LIN {X 0,Y 256.355,Z 531.803,A -85,B 0,C 180,E1 -21459.86,E2 -21459.86} C_VEL
LIN {X 0,Y 252.646,Z 547.764,A -85,B 0,C 180,E1 -21461.014,E2 -21461.014} C_VEL
LIN {X 0,Y 248.399,Z 562.44,A -85,B 0,C 180,E1 -21462.341,E2 -21462.341} C_VEL
LIN {X 0,Y 243.325,Z 577.415,A -85,B 0,C 180,E1 -21464.072,E2 -21464.072} C_VEL
LIN {X 0,Y 238.018,Z 591.108,A -85,B 0,C 180,E1 -21466.062,E2 -21466.062} C_VEL
LIN {X 0,Y 233.373,Z 601.837,A -85,B 0,C 180,E1 -21467.929,E2 -21467.929} C_VEL
LIN {X 0,Y 227.446,Z 614.36,A -85,B 0,C 180,E1 -21470.578,E2 -21470.578} C_VEL
LIN {X 0,Y 221.787,Z 625.54,A -85,B 0,C 180,E1 -21473.548,E2 -21473.548} C_VEL
LIN {X 0,Y 216.728,Z 634.804,A -85,B 0,C 180,E1 -21476.546,E2 -21476.546} C_VEL
LIN {X 0,Y 211.759,Z 643.811,A -85,B 0,C 180,E1 -21480.144,E2 -21480.144} C_VEL
LIN {X 0,Y 207.469,Z 651.338,A -85,B 0,C 180,E1 -21483.872,E2 -21483.872} C_VEL
LIN {X 0,Y 204.013,Z 657.483,A -85,B 0,C 180,E1 -21487.732,E2 -21487.732} C_VEL
LIN {X 0,Y 201.336,Z 662.513,A -85,B 0,C 180,E1 -21491.69,E2 -21491.69} C_VEL
LIN {X 0,Y 199.353,Z 666.403,A -85,B 0,C 180,E1 -21495.713,E2 -21495.713} C_VEL
LIN {X 0,Y 198.192,Z 669.285,A -85,B 0,C 180,E1 -21499.787,E2 -21499.787} C_VEL
LIN {X 0,Y 197.545,Z 671.175,A -85,B 0,C 180,E1 -21503.873,E2 -21503.873} C_VEL
LIN {X 0,Y 197.351,Z 672.126,A -85,B 0,C 180,E1 -21507.959,E2 -21507.959} C_VEL
LIN {X 0,Y 197.395,Z 672.279,A -85,B 0,C 180,E1 -21510,E2 -21510} C_VEL
LIN {X 0,Y 197.415,Z 671.675,A -85,B 0,C 180,E1 -21514.579,E2 -21514.579} C_VEL
LIN {X 0,Y 197.782,Z 670.45,A -85,B 0,C 180,E1 -21518.171,E2 -21518.171} C_VEL
LIN {X 0,Y 198.684,Z 668.056,A -85,B 0,C 180,E1 -21522.253,E2 -21522.253} C_VEL
LIN {X 0,Y 200.261,Z 664.751,A -85,B 0,C 180,E1 -21526.305,E2 -21526.305} C_VEL
LIN {X 0,Y 203.161,Z 659.194,A -85,B 0,C 180,E1 -21531.192,E2 -21531.192} C_VEL
LIN {X 0,Y 207.427,Z 651.578,A -85,B 0,C 180,E1 -21536.133,E2 -21536.133} C_VEL
LIN {X 0,Y 212.494,Z 642.647,A -85,B 0,C 180,E1 -21540.524,E2 -21540.524} C_VEL
LIN {X 0,Y 217.342,Z 633.912,A -85,B 0,C 180,E1 -21543.903,E2 -21543.903} C_VEL
LIN {X 0,Y 222.404,Z 624.465,A -85,B 0,C 180,E1 -21546.898,E2 -21546.898} C_VEL
LIN {X 0,Y 227.991,Z 613.516,A -85,B 0,C 180,E1 -21549.74,E2 -21549.74} C_VEL
LIN {X 0,Y 234.118,Z 600.392,A -85,B 0,C 180,E1 -21552.487,E2 -21552.487} C_VEL
LIN {X 0,Y 240.281,Z 586.013,A -85,B 0,C 180,E1 -21554.847,E2 -21554.847} C_VEL
LIN {X 0,Y 245.182,Z 572.494,A -85,B 0,C 180,E1 -21556.664,E2 -21556.664} C_VEL
LIN {X 0,Y 249.822,Z 558.149,A -85,B 0,C 180,E1 -21558.201,E2 -21558.201} C_VEL
LIN {X 0,Y 254.135,Z 542.579,A -85,B 0,C 180,E1 -21559.508,E2 -21559.508} C_VEL
LIN {X 0,Y 257.325,Z 527.974,A -85,B 0,C 180,E1 -21560.493,E2 -21560.493} C_VEL
LIN {X 0,Y 259.966,Z 512.67,A -85,B 0,C 180,E1 -21561.239,E2 -21561.239} C_VEL
LIN {X 0,Y 261.928,Z 495.841,A -85,B 0,C 180,E1 -21561.832,E2 -21561.832} C_VEL
LIN {X 0,Y 268.666,Z 399.885,A -85,B 0,C 180,E1 -21564.176,E2 -21564.176} C_VEL
LIN {X 0,Y 261.466,Z 386.886,A -85,B 0,C 180,E1 -21567.08,E2 -21567.08} C_VEL
LIN {X 0,Y 255.056,Z 376.394,A -85,B 0,C 180,E1 -21569.969,E2 -21569.969} C_VEL
LIN {X 0,Y 249.229,Z 367.595,A -85,B 0,C 180,E1 -21572.938,E2 -21572.938} C_VEL
LIN {X 0,Y 243.586,Z 359.592,A -85,B 0,C 180,E1 -21576.259,E2 -21576.259} C_VEL
LIN {X 0,Y 240.202,Z 355.081,A -85,B 0,C 180,E1 -21578.547,E2 -21578.547} C_VEL
LIN {X 0,Y 237.313,Z 351.233,A -85,B 0,C 180,E1 -21580.763,E2 -21580.763} C_VEL
LIN {X 0,Y 233.816,Z 346.937,A -85,B 0,C 180,E1 -21583.889,E2 -21583.889} C_VEL
LIN {X 0,Y 233.178,Z 345.639,A -85,B 0,C 180,E1 -21584.597,E2 -21584.597} C_VEL
LIN {X 0,Y 230.388,Z 342.989,A -85,B 0,C 180,E1 -21587.782,E2 -21587.782} C_VEL
LIN {X 0,Y 229.018,Z 340.216,A -85,B 0,C 180,E1 -21590,E2 -21590} C_VEL
LIN {X 0,Y 226.04,Z 337.167,A -85,B 0,C 180,E1 -21600,E2 -21600} C_VEL
LIN {X 0,Y 229.187,Z 340.456,A -85,B 0,C 180,E1 -21609.918,E2 -21609.918} C_VEL
LIN {X 0,Y 230.98,Z 343.781,A -85,B 0,C 180,E1 -21612.632,E2 -21612.632} C_VEL
LIN {X 0,Y 231.708,Z 344.547,A -85,B 0,C 180,E1 -21613.5,E2 -21613.5} C_VEL
LIN {X 0,Y 232.852,Z 346.488,A -85,B 0,C 180,E1 -21614.84,E2 -21614.84} C_VEL
LIN {X 0,Y 233.872,Z 349.492,A -85,B 0,C 180,E1 -21616.07,E2 -21616.07} C_VEL
LIN {X 0,Y 236.74,Z 358.879,A -85,B 0,C 180,E1 -21619.163,E2 -21619.163} C_VEL
LIN {X 0,Y 237.715,Z 360.77,A -85,B 0,C 180,E1 -21619.984,E2 -21619.984} C_VEL
LIN {X 0,Y 239.314,Z 362.778,A -85,B 0,C 180,E1 -21621.165,E2 -21621.165} C_VEL
LIN {X 0,Y 242.766,Z 367.633,A -85,B 0,C 180,E1 -21623.513,E2 -21623.513} C_VEL
LIN {X 0,Y 247.755,Z 374.869,A -85,B 0,C 180,E1 -21626.48,E2 -21626.48} C_VEL
LIN {X 0,Y 250.61,Z 379.612,A -85,B 0,C 180,E1 -21628.035,E2 -21628.035} C_VEL
LIN {X 0,Y 254.986,Z 387.886,A -85,B 0,C 180,E1 -21630.269,E2 -21630.269} C_VEL
LIN {X 0,Y 259.314,Z 396.661,A -85,B 0,C 180,E1 -21632.304,E2 -21632.304} C_VEL
LIN {X 0,Y 264.179,Z 407.344,A -85,B 0,C 180,E1 -21634.43,E2 -21634.43} C_VEL
LIN {X 0,Y 256.78,Z 508.197,A -85,B 0,C 180,E1 -21636.898,E2 -21636.898} C_VEL
LIN {X 0,Y 254.514,Z 524.569,A -85,B 0,C 180,E1 -21637.486,E2 -21637.486} C_VEL
LIN {X 0,Y 251.376,Z 540.299,A -85,B 0,C 180,E1 -21638.254,E2 -21638.254} C_VEL
LIN {X 0,Y 247.487,Z 555.955,A -85,B 0,C 180,E1 -21639.302,E2 -21639.302} C_VEL
LIN {X 0,Y 242.994,Z 570.902,A -85,B 0,C 180,E1 -21640.606,E2 -21640.606} C_VEL
LIN {X 0,Y 237.526,Z 586.138,A -85,B 0,C 180,E1 -21642.294,E2 -21642.294} C_VEL
LIN {X 0,Y 232.084,Z 599.431,A -85,B 0,C 180,E1 -21644.145,E2 -21644.145} C_VEL
LIN {X 0,Y 226.38,Z 612.043,A -85,B 0,C 180,E1 -21646.311,E2 -21646.311} C_VEL
LIN {X 0,Y 220.841,Z 623.266,A -85,B 0,C 180,E1 -21648.674,E2 -21648.674} C_VEL
LIN {X 0,Y 214.91,Z 634.459,A -85,B 0,C 180,E1 -21651.587,E2 -21651.587} C_VEL
LIN {X 0,Y 209.666,Z 644.078,A -85,B 0,C 180,E1 -21654.675,E2 -21654.675} C_VEL
LIN {X 0,Y 204.309,Z 653.434,A -85,B 0,C 180,E1 -21658.36,E2 -21658.36} C_VEL
LIN {X 0,Y 199.292,Z 662.116,A -85,B 0,C 180,E1 -21662.714,E2 -21662.714} C_VEL
LIN {X 0,Y 195.109,Z 669.816,A -85,B 0,C 180,E1 -21667.777,E2 -21667.777} C_VEL
LIN {X 0,Y 192.308,Z 675.69,A -85,B 0,C 180,E1 -21673.001,E2 -21673.001} C_VEL
LIN {X 0,Y 190.824,Z 679.128,A -85,B 0,C 180,E1 -21677.234,E2 -21677.234} C_VEL
LIN {X 0,Y 190.209,Z 681.639,A -85,B 0,C 180,E1 -21681.501,E2 -21681.501} C_VEL
LIN {X 0,Y 190.132,Z 683.209,A -85,B 0,C 180,E1 -21686.391,E2 -21686.391} C_VEL
LIN {X 0,Y 190.266,Z 683.598,A -85,B 0,C 180,E1 -21690,E2 -21690} C_VEL
LIN {X 0,Y 190.135,Z 683.05,A -85,B 0,C 180,E1 -21694.24,E2 -21694.24} C_VEL
LIN {X 0,Y 190.209,Z 681.613,A -85,B 0,C 180,E1 -21698.499,E2 -21698.499} C_VEL
LIN {X 0,Y 190.822,Z 679.09,A -85,B 0,C 180,E1 -21702.767,E2 -21702.767} C_VEL
LIN {X 0,Y 192.305,Z 675.638,A -85,B 0,C 180,E1 -21707,E2 -21707} C_VEL
LIN {X 0,Y 195.11,Z 669.748,A -85,B 0,C 180,E1 -21712.223,E2 -21712.223} C_VEL
LIN {X 0,Y 199.333,Z 662.022,A -85,B 0,C 180,E1 -21717.28,E2 -21717.28} C_VEL
LIN {X 0,Y 204.316,Z 653.323,A -85,B 0,C 180,E1 -21721.639,E2 -21721.639} C_VEL
LIN {X 0,Y 209.695,Z 643.944,A -85,B 0,C 180,E1 -21725.32,E2 -21725.32} C_VEL
LIN {X 0,Y 214.905,Z 634.295,A -85,B 0,C 180,E1 -21728.415,E2 -21728.415} C_VEL
LIN {X 0,Y 220.799,Z 623.063,A -85,B 0,C 180,E1 -21731.335,E2 -21731.335} C_VEL
LIN {X 0,Y 226.838,Z 610.839,A -85,B 0,C 180,E1 -21733.886,E2 -21733.886} C_VEL
LIN {X 0,Y 232.597,Z 597.907,A -85,B 0,C 180,E1 -21736.056,E2 -21736.056} C_VEL
LIN {X 0,Y 238.044,Z 584.374,A -85,B 0,C 180,E1 -21737.884,E2 -21737.884} C_VEL
LIN {X 0,Y 242.967,Z 570.483,A -85,B 0,C 180,E1 -21739.402,E2 -21739.402} C_VEL
LIN {X 0,Y 247.766,Z 554.474,A -85,B 0,C 180,E1 -21740.78,E2 -21740.78} C_VEL
LIN {X 0,Y 251.355,Z 539.708,A -85,B 0,C 180,E1 -21741.75,E2 -21741.75} C_VEL
LIN {X 0,Y 254.473,Z 523.669,A -85,B 0,C 180,E1 -21742.53,E2 -21742.53} C_VEL
LIN {X 0,Y 256.608,Z 508.275,A -85,B 0,C 180,E1 -21743.071,E2 -21743.071} C_VEL
LIN {X 0,Y 264.022,Z 407.323,A -85,B 0,C 180,E1 -21745.54,E2 -21745.54} C_VEL
LIN {X 0,Y 258.866,Z 395.777,A -85,B 0,C 180,E1 -21747.805,E2 -21747.805} C_VEL
LIN {X 0,Y 252.961,Z 384.159,A -85,B 0,C 180,E1 -21750.624,E2 -21750.624} C_VEL
LIN {X 0,Y 248.839,Z 376.699,A -85,B 0,C 180,E1 -21752.795,E2 -21752.795} C_VEL
LIN {X 0,Y 243.953,Z 369.435,A -85,B 0,C 180,E1 -21755.593,E2 -21755.593} C_VEL
LIN {X 0,Y 240.843,Z 365.015,A -85,B 0,C 180,E1 -21757.592,E2 -21757.592} C_VEL
LIN {X 0,Y 238.229,Z 361.399,A -85,B 0,C 180,E1 -21759.45,E2 -21759.45} C_VEL
LIN {X 0,Y 235.016,Z 357.028,A -85,B 0,C 180,E1 -21762.038,E2 -21762.038} C_VEL
LIN {X 0,Y 232.253,Z 353.396,A -85,B 0,C 180,E1 -21764.647,E2 -21764.647} C_VEL
LIN {X 0,Y 231.47,Z 352.253,A -85,B 0,C 180,E1 -21765.494,E2 -21765.494} C_VEL
LIN {X 0,Y 228.798,Z 349.202,A -85,B 0,C 180,E1 -21768.764,E2 -21768.764} C_VEL
LIN {X 0,Y 227.904,Z 347.196,A -85,B 0,C 180,E1 -21770.282,E2 -21770.282} C_VEL
LIN {X 0,Y 224.916,Z 343.654,A -85,B 0,C 180,E1 -21780,E2 -21780} C_VEL
LIN {X 0,Y 228.009,Z 347.425,A -85,B 0,C 180,E1 -21790.363,E2 -21790.363} C_VEL
LIN {X 0,Y 229.777,Z 350.617,A -85,B 0,C 180,E1 -21793.037,E2 -21793.037} C_VEL
LIN {X 0,Y 231.866,Z 352.688,A -85,B 0,C 180,E1 -21795.38,E2 -21795.38} C_VEL
LIN {X 0,Y 234.403,Z 356.438,A -85,B 0,C 180,E1 -21797.898,E2 -21797.898} C_VEL
LIN {X 0,Y 235.676,Z 357.892,A -85,B 0,C 180,E1 -21798.98,E2 -21798.98} C_VEL
LIN {X 0,Y 239.348,Z 362.897,A -85,B 0,C 180,E1 -21801.821,E2 -21801.821} C_VEL
LIN {X 0,Y 242.557,Z 367.481,A -85,B 0,C 180,E1 -21803.994,E2 -21803.994} C_VEL
LIN {X 0,Y 247.648,Z 374.78,A -85,B 0,C 180,E1 -21807.005,E2 -21807.005} C_VEL
LIN {X 0,Y 253.24,Z 383.624,A -85,B 0,C 180,E1 -21809.913,E2 -21809.913} C_VEL
LIN {X 0,Y 259.105,Z 393.578,A -85,B 0,C 180,E1 -21812.622,E2 -21812.622} C_VEL
LIN {X 0,Y 264.235,Z 403.101,A -85,B 0,C 180,E1 -21814.785,E2 -21814.785} C_VEL
LIN {X 0,Y 257.124,Z 499.809,A -85,B 0,C 180,E1 -21817.158,E2 -21817.158} C_VEL
LIN {X 0,Y 254.847,Z 516.467,A -85,B 0,C 180,E1 -21817.79,E2 -21817.79} C_VEL
LIN {X 0,Y 251.866,Z 532.019,A -85,B 0,C 180,E1 -21818.62,E2 -21818.62} C_VEL
LIN {X 0,Y 248.049,Z 547.978,A -85,B 0,C 180,E1 -21819.778,E2 -21819.778} C_VEL
LIN {X 0,Y 243.661,Z 562.653,A -85,B 0,C 180,E1 -21821.103,E2 -21821.103} C_VEL
LIN {X 0,Y 238.542,Z 577.273,A -85,B 0,C 180,E1 -21822.795,E2 -21822.795} C_VEL
LIN {X 0,Y 232.937,Z 591.32,A -85,B 0,C 180,E1 -21824.845,E2 -21824.845} C_VEL
LIN {X 0,Y 228.13,Z 602.048,A -85,B 0,C 180,E1 -21826.729,E2 -21826.729} C_VEL
LIN {X 0,Y 222.235,Z 614.078,A -85,B 0,C 180,E1 -21829.294,E2 -21829.294} C_VEL
LIN {X 0,Y 216.053,Z 625.752,A -85,B 0,C 180,E1 -21832.416,E2 -21832.416} C_VEL
LIN {X 0,Y 210.794,Z 635.015,A -85,B 0,C 180,E1 -21835.474,E2 -21835.474} C_VEL
LIN {X 0,Y 206.351,Z 642.704,A -85,B 0,C 180,E1 -21838.539,E2 -21838.539} C_VEL
LIN {X 0,Y 202.098,Z 649.76,A -85,B 0,C 180,E1 -21842.001,E2 -21842.001} C_VEL
LIN {X 0,Y 198.235,Z 656.288,A -85,B 0,C 180,E1 -21845.939,E2 -21845.939} C_VEL
LIN {X 0,Y 195.195,Z 661.564,A -85,B 0,C 180,E1 -21849.998,E2 -21849.998} C_VEL
LIN {X 0,Y 193.445,Z 664.821,A -85,B 0,C 180,E1 -21853.103,E2 -21853.103} C_VEL
LIN {X 0,Y 191.726,Z 668.166,A -85,B 0,C 180,E1 -21857.295,E2 -21857.295} C_VEL
LIN {X 0,Y 190.739,Z 670.591,A -85,B 0,C 180,E1 -21861.525,E2 -21861.525} C_VEL
LIN {X 0,Y 190.316,Z 671.962,A -85,B 0,C 180,E1 -21865.764,E2 -21865.764} C_VEL
LIN {X 0,Y 190.299,Z 672.486,A -85,B 0,C 180,E1 -21870,E2 -21870} C_VEL
LIN {X 0,Y 190.336,Z 671.943,A -85,B 0,C 180,E1 -21874.473,E2 -21874.473} C_VEL
LIN {X 0,Y 190.735,Z 670.657,A -85,B 0,C 180,E1 -21878.475,E2 -21878.475} C_VEL
LIN {X 0,Y 191.698,Z 668.265,A -85,B 0,C 180,E1 -21882.707,E2 -21882.707} C_VEL
LIN {X 0,Y 193.393,Z 664.96,A -85,B 0,C 180,E1 -21886.901,E2 -21886.901} C_VEL
LIN {X 0,Y 196.509,Z 659.402,A -85,B 0,C 180,E1 -21891.946,E2 -21891.946} C_VEL
LIN {X 0,Y 201.025,Z 651.786,A -85,B 0,C 180,E1 -21897.032,E2 -21897.032} C_VEL
LIN {X 0,Y 205.474,Z 644.292,A -85,B 0,C 180,E1 -21900.867,E2 -21900.867} C_VEL
LIN {X 0,Y 210.718,Z 635.341,A -85,B 0,C 180,E1 -21904.541,E2 -21904.541} C_VEL
LIN {X 0,Y 216.73,Z 624.671,A -85,B 0,C 180,E1 -21908.033,E2 -21908.033} C_VEL
LIN {X 0,Y 222.015,Z 614.783,A -85,B 0,C 180,E1 -21910.666,E2 -21910.666} C_VEL
LIN {X 0,Y 227.999,Z 602.563,A -85,B 0,C 180,E1 -21913.302,E2 -21913.302} C_VEL
LIN {X 0,Y 233.836,Z 589.598,A -85,B 0,C 180,E1 -21915.545,E2 -21915.545} C_VEL
LIN {X 0,Y 239.245,Z 575.678,A -85,B 0,C 180,E1 -21917.535,E2 -21917.535} C_VEL
LIN {X 0,Y 244.103,Z 561.867,A -85,B 0,C 180,E1 -21919.092,E2 -21919.092} C_VEL
LIN {X 0,Y 248.782,Z 546.044,A -85,B 0,C 180,E1 -21920.494,E2 -21920.494} C_VEL
LIN {X 0,Y 252.312,Z 530.768,A -85,B 0,C 180,E1 -21921.573,E2 -21921.573} C_VEL
LIN {X 0,Y 255.283,Z 514.695,A -85,B 0,C 180,E1 -21922.405,E2 -21922.405} C_VEL
LIN {X 0,Y 257.404,Z 498.341,A -85,B 0,C 180,E1 -21923.007,E2 -21923.007} C_VEL
LIN {X 0,Y 264.379,Z 403.201,A -85,B 0,C 180,E1 -21925.336,E2 -21925.336} C_VEL
LIN {X 0,Y 257.937,Z 391.337,A -85,B 0,C 180,E1 -21928.089,E2 -21928.089} C_VEL
LIN {X 0,Y 251.758,Z 381.087,A -85,B 0,C 180,E1 -21931.031,E2 -21931.031} C_VEL
LIN {X 0,Y 246.279,Z 372.741,A -85,B 0,C 180,E1 -21933.986,E2 -21933.986} C_VEL
LIN {X 0,Y 241.405,Z 365.667,A -85,B 0,C 180,E1 -21937.016,E2 -21937.016} C_VEL
LIN {X 0,Y 238.371,Z 361.458,A -85,B 0,C 180,E1 -21939.167,E2 -21939.167} C_VEL
LIN {X 0,Y 235.618,Z 357.627,A -85,B 0,C 180,E1 -21941.382,E2 -21941.382} C_VEL
LIN {X 0,Y 232.556,Z 353.86,A -85,B 0,C 180,E1 -21944.217,E2 -21944.217} C_VEL
LIN {X 0,Y 231.597,Z 352.309,A -85,B 0,C 180,E1 -21945.277,E2 -21945.277} C_VEL
LIN {X 0,Y 228.989,Z 349.446,A -85,B 0,C 180,E1 -21948.492,E2 -21948.492} C_VEL
LIN {X 0,Y 227.978,Z 347.193,A -85,B 0,C 180,E1 -21950.251,E2 -21950.251} C_VEL
LIN {X 0,Y 225.174,Z 344.216,A -85,B 0,C 180,E1 -21960,E2 -21960} C_VEL
LIN {X 0,Y 228.071,Z 347.38,A -85,B 0,C 180,E1 -21969.555,E2 -21969.555} C_VEL
LIN {X 0,Y 229.858,Z 350.729,A -85,B 0,C 180,E1 -21972.358,E2 -21972.358} C_VEL
LIN {X 0,Y 232.01,Z 352.846,A -85,B 0,C 180,E1 -21974.808,E2 -21974.808} C_VEL
LIN {X 0,Y 234.641,Z 356.671,A -85,B 0,C 180,E1 -21977.428,E2 -21977.428} C_VEL
LIN {X 0,Y 235.785,Z 357.977,A -85,B 0,C 180,E1 -21978.407,E2 -21978.407} C_VEL
LIN {X 0,Y 237.715,Z 360.77,A -85,B 0,C 180,E1 -21979.984,E2 -21979.984} C_VEL
LIN {X 0,Y 239.155,Z 363.83,A -85,B 0,C 180,E1 -21981.152,E2 -21981.152} C_VEL
LIN {X 0,Y 243.386,Z 377.192,A -85,B 0,C 180,E1 -21984.513,E2 -21984.513} C_VEL
LIN {X 0,Y 245.148,Z 380.425,A -85,B 0,C 180,E1 -21985.608,E2 -21985.608} C_VEL
LIN {X 0,Y 248.213,Z 385.624,A -85,B 0,C 180,E1 -21987.356,E2 -21987.356} C_VEL
LIN {X 0,Y 252.446,Z 393.909,A -85,B 0,C 180,E1 -21989.614,E2 -21989.614} C_VEL
LIN {X 0,Y 256.868,Z 403.281,A -85,B 0,C 180,E1 -21991.781,E2 -21991.781} C_VEL
LIN {X 0,Y 260.029,Z 410.421,A -85,B 0,C 180,E1 -21993.233,E2 -21993.233} C_VEL
LIN {X 0,Y 252.581,Z 508.008,A -85,B 0,C 180,E1 -21995.61,E2 -21995.61} C_VEL
LIN {X 0,Y 250.219,Z 524.616,A -85,B 0,C 180,E1 -21996.207,E2 -21996.207} C_VEL
LIN {X 0,Y 247.007,Z 540.242,A -85,B 0,C 180,E1 -21996.968,E2 -21996.968} C_VEL
LIN {X 0,Y 243.045,Z 555.754,A -85,B 0,C 180,E1 -21998.004,E2 -21998.004} C_VEL
LIN {X 0,Y 238.425,Z 570.7,A -85,B 0,C 180,E1 -21999.308,E2 -21999.308} C_VEL
LIN {X 0,Y 232.785,Z 585.934,A -85,B 0,C 180,E1 -22000.995,E2 -22000.995} C_VEL
LIN {X 0,Y 227.61,Z 598.262,A -85,B 0,C 180,E1 -22002.707,E2 -22002.707} C_VEL
LIN {X 0,Y 221.274,Z 611.838,A -85,B 0,C 180,E1 -22005.034,E2 -22005.034} C_VEL
LIN {X 0,Y 215.475,Z 623.058,A -85,B 0,C 180,E1 -22007.407,E2 -22007.407} C_VEL
LIN {X 0,Y 209.31,Z 634.251,A -85,B 0,C 180,E1 -22010.361,E2 -22010.361} C_VEL
LIN {X 0,Y 203.856,Z 643.87,A -85,B 0,C 180,E1 -22013.509,E2 -22013.509} C_VEL
LIN {X 0,Y 198.192,Z 653.225,A -85,B 0,C 180,E1 -22017.264,E2 -22017.264} C_VEL
LIN {X 0,Y 192.898,Z 661.906,A -85,B 0,C 180,E1 -22021.73,E2 -22021.73} C_VEL
LIN {X 0,Y 188.435,Z 669.606,A -85,B 0,C 180,E1 -22026.945,E2 -22026.945} C_VEL
LIN {X 0,Y 185.452,Z 675.481,A -85,B 0,C 180,E1 -22032.352,E2 -22032.352} C_VEL
LIN {X 0,Y 183.829,Z 678.919,A -85,B 0,C 180,E1 -22036.739,E2 -22036.739} C_VEL
LIN {X 0,Y 183.147,Z 681.431,A -85,B 0,C 180,E1 -22041.171,E2 -22041.171} C_VEL
LIN {X 0,Y 183.032,Z 683.099,A -85,B 0,C 180,E1 -22046.688,E2 -22046.688} C_VEL
LIN {X 0,Y 183.171,Z 683.391,A -85,B 0,C 180,E1 -22050,E2 -22050} C_VEL
LIN {X 0,Y 183.031,Z 682.842,A -85,B 0,C 180,E1 -22054.404,E2 -22054.404} C_VEL
LIN {X 0,Y 183.147,Z 681.404,A -85,B 0,C 180,E1 -22058.829,E2 -22058.829} C_VEL
LIN {X 0,Y 183.827,Z 678.88,A -85,B 0,C 180,E1 -22063.261,E2 -22063.261} C_VEL
LIN {X 0,Y 185.45,Z 675.428,A -85,B 0,C 180,E1 -22067.648,E2 -22067.648} C_VEL
LIN {X 0,Y 188.436,Z 669.536,A -85,B 0,C 180,E1 -22073.055,E2 -22073.055} C_VEL
LIN {X 0,Y 192.942,Z 661.81,A -85,B 0,C 180,E1 -22078.264,E2 -22078.264} C_VEL
LIN {X 0,Y 198.2,Z 653.111,A -85,B 0,C 180,E1 -22082.735,E2 -22082.735} C_VEL
LIN {X 0,Y 203.869,Z 643.732,A -85,B 0,C 180,E1 -22086.488,E2 -22086.488} C_VEL
LIN {X 0,Y 209.313,Z 634.082,A -85,B 0,C 180,E1 -22089.639,E2 -22089.639} C_VEL
LIN {X 0,Y 215.461,Z 622.85,A -85,B 0,C 180,E1 -22092.596,E2 -22092.596} C_VEL
LIN {X 0,Y 221.742,Z 610.627,A -85,B 0,C 180,E1 -22095.167,E2 -22095.167} C_VEL
LIN {X 0,Y 227.724,Z 597.627,A -85,B 0,C 180,E1 -22097.362,E2 -22097.362} C_VEL
LIN {X 0,Y 233.311,Z 584.161,A -85,B 0,C 180,E1 -22099.186,E2 -22099.186} C_VEL
LIN {X 0,Y 238.38,Z 570.269,A -85,B 0,C 180,E1 -22100.706,E2 -22100.706} C_VEL
LIN {X 0,Y 243.325,Z 554.26,A -85,B 0,C 180,E1 -22102.08,E2 -22102.08} C_VEL
LIN {X 0,Y 246.967,Z 539.717,A -85,B 0,C 180,E1 -22103.031,E2 -22103.031} C_VEL
LIN {X 0,Y 250.298,Z 522.99,A -85,B 0,C 180,E1 -22103.837,E2 -22103.837} C_VEL
LIN {X 0,Y 252.404,Z 508.049,A -85,B 0,C 180,E1 -22104.36,E2 -22104.36} C_VEL
LIN {X 0,Y 259.858,Z 410.263,A -85,B 0,C 180,E1 -22106.745,E2 -22106.745} C_VEL
LIN {X 0,Y 254.28,Z 397.834,A -85,B 0,C 180,E1 -22109.36,E2 -22109.36} C_VEL
LIN {X 0,Y 249.79,Z 388.827,A -85,B 0,C 180,E1 -22111.655,E2 -22111.655} C_VEL
LIN {X 0,Y 246.4,Z 382.544,A -85,B 0,C 180,E1 -22113.534,E2 -22113.534} C_VEL
LIN {X 0,Y 241.818,Z 375.583,A -85,B 0,C 180,E1 -22116.275,E2 -22116.275} C_VEL
LIN {X 0,Y 239.091,Z 371.578,A -85,B 0,C 180,E1 -22118.103,E2 -22118.103} C_VEL
LIN {X 0,Y 236.501,Z 367.876,A -85,B 0,C 180,E1 -22120.017,E2 -22120.017} C_VEL
LIN {X 0,Y 233.435,Z 363.613,A -85,B 0,C 180,E1 -22122.592,E2 -22122.592} C_VEL
LIN {X 0,Y 230.665,Z 359.733,A -85,B 0,C 180,E1 -22125.357,E2 -22125.357} C_VEL
LIN {X 0,Y 229.633,Z 358.605,A -85,B 0,C 180,E1 -22126.505,E2 -22126.505} C_VEL
LIN {X 0,Y 227.336,Z 355.405,A -85,B 0,C 180,E1 -22129.649,E2 -22129.649} C_VEL
LIN {X 0,Y 226.798,Z 354.13,A -85,B 0,C 180,E1 -22130.637,E2 -22130.637} C_VEL
LIN {X 0,Y 224.049,Z 350.715,A -85,B 0,C 180,E1 -22140,E2 -22140} C_VEL
LIN {X 0,Y 226.876,Z 354.311,A -85,B 0,C 180,E1 -22149.969,E2 -22149.969} C_VEL
LIN {X 0,Y 228.742,Z 357.651,A -85,B 0,C 180,E1 -22152.871,E2 -22152.871} C_VEL
LIN {X 0,Y 230.593,Z 359.602,A -85,B 0,C 180,E1 -22155.015,E2 -22155.015} C_VEL
LIN {X 0,Y 233.076,Z 363.27,A -85,B 0,C 180,E1 -22157.55,E2 -22157.55} C_VEL
LIN {X 0,Y 234.221,Z 364.696,A -85,B 0,C 180,E1 -22158.563,E2 -22158.563} C_VEL
LIN {X 0,Y 237.68,Z 369.544,A -85,B 0,C 180,E1 -22161.334,E2 -22161.334} C_VEL
LIN {X 0,Y 240.869,Z 374.233,A -85,B 0,C 180,E1 -22163.568,E2 -22163.568} C_VEL
LIN {X 0,Y 244.172,Z 379.153,A -85,B 0,C 180,E1 -22165.636,E2 -22165.636} C_VEL
LIN {X 0,Y 249.435,Z 387.31,A -85,B 0,C 180,E1 -22168.561,E2 -22168.561} C_VEL
LIN {X 0,Y 255.817,Z 398.386,A -85,B 0,C 180,E1 -22171.696,E2 -22171.696} C_VEL
LIN {X 0,Y 260.013,Z 406.349,A -85,B 0,C 180,E1 -22173.57,E2 -22173.57} C_VEL
LIN {X 0,Y 253.02,Z 498.801,A -85,B 0,C 180,E1 -22175.843,E2 -22175.843} C_VEL
LIN {X 0,Y 250.878,Z 514.856,A -85,B 0,C 180,E1 -22176.437,E2 -22176.437} C_VEL
LIN {X 0,Y 247.803,Z 530.938,A -85,B 0,C 180,E1 -22177.261,E2 -22177.261} C_VEL
LIN {X 0,Y 244.129,Z 546.213,A -85,B 0,C 180,E1 -22178.328,E2 -22178.328} C_VEL
LIN {X 0,Y 239.592,Z 561.158,A -85,B 0,C 180,E1 -22179.647,E2 -22179.647} C_VEL
LIN {X 0,Y 234.636,Z 575.144,A -85,B 0,C 180,E1 -22181.221,E2 -22181.221} C_VEL
LIN {X 0,Y 228.988,Z 589.197,A -85,B 0,C 180,E1 -22183.204,E2 -22183.204} C_VEL
LIN {X 0,Y 223.453,Z 601.288,A -85,B 0,C 180,E1 -22185.273,E2 -22185.273} C_VEL
LIN {X 0,Y 217.482,Z 613.098,A -85,B 0,C 180,E1 -22187.789,E2 -22187.789} C_VEL
LIN {X 0,Y 211.254,Z 624.489,A -85,B 0,C 180,E1 -22190.796,E2 -22190.796} C_VEL
LIN {X 0,Y 204.95,Z 635.225,A -85,B 0,C 180,E1 -22194.342,E2 -22194.342} C_VEL
LIN {X 0,Y 199.432,Z 644.234,A -85,B 0,C 180,E1 -22198.089,E2 -22198.089} C_VEL
LIN {X 0,Y 194.694,Z 651.759,A -85,B 0,C 180,E1 -22202.013,E2 -22202.013} C_VEL
LIN {X 0,Y 190.004,Z 659.308,A -85,B 0,C 180,E1 -22207.146,E2 -22207.146} C_VEL
LIN {X 0,Y 186.606,Z 665.031,A -85,B 0,C 180,E1 -22212.464,E2 -22212.464} C_VEL
LIN {X 0,Y 184.761,Z 668.375,A -85,B 0,C 180,E1 -22216.807,E2 -22216.807} C_VEL
LIN {X 0,Y 183.716,Z 670.799,A -85,B 0,C 180,E1 -22221.198,E2 -22221.198} C_VEL
LIN {X 0,Y 183.221,Z 672.211,A -85,B 0,C 180,E1 -22225.798,E2 -22225.798} C_VEL
LIN {X 0,Y 183.205,Z 672.693,A -85,B 0,C 180,E1 -22230,E2 -22230} C_VEL
LIN {X 0,Y 183.232,Z 672.202,A -85,B 0,C 180,E1 -22234.399,E2 -22234.399} C_VEL
LIN {X 0,Y 183.711,Z 670.864,A -85,B 0,C 180,E1 -22238.802,E2 -22238.802} C_VEL
LIN {X 0,Y 184.735,Z 668.473,A -85,B 0,C 180,E1 -22243.195,E2 -22243.195} C_VEL
LIN {X 0,Y 186.557,Z 665.168,A -85,B 0,C 180,E1 -22247.54,E2 -22247.54} C_VEL
LIN {X 0,Y 189.95,Z 659.484,A -85,B 0,C 180,E1 -22252.86,E2 -22252.86} C_VEL
LIN {X 0,Y 194.656,Z 651.994,A -85,B 0,C 180,E1 -22257.992,E2 -22257.992} C_VEL
LIN {X 0,Y 199.342,Z 644.5,A -85,B 0,C 180,E1 -22261.927,E2 -22261.927} C_VEL
LIN {X 0,Y 204.874,Z 635.547,A -85,B 0,C 180,E1 -22265.673,E2 -22265.673} C_VEL
LIN {X 0,Y 211.146,Z 624.877,A -85,B 0,C 180,E1 -22269.228,E2 -22269.228} C_VEL
LIN {X 0,Y 217.313,Z 613.704,A -85,B 0,C 180,E1 -22272.201,E2 -22272.201} C_VEL
LIN {X 0,Y 223.785,Z 600.802,A -85,B 0,C 180,E1 -22274.96,E2 -22274.96} C_VEL
LIN {X 0,Y 229.924,Z 587.467,A -85,B 0,C 180,E1 -22277.188,E2 -22277.188} C_VEL
LIN {X 0,Y 234.562,Z 575.736,A -85,B 0,C 180,E1 -22278.833,E2 -22278.833} C_VEL
LIN {X 0,Y 239.501,Z 562.069,A -85,B 0,C 180,E1 -22280.379,E2 -22280.379} C_VEL
LIN {X 0,Y 244.328,Z 546.245,A -85,B 0,C 180,E1 -22281.778,E2 -22281.778} C_VEL
LIN {X 0,Y 247.692,Z 532.263,A -85,B 0,C 180,E1 -22282.772,E2 -22282.772} C_VEL
LIN {X 0,Y 250.731,Z 516.718,A -85,B 0,C 180,E1 -22283.608,E2 -22283.608} C_VEL
LIN {X 0,Y 253.025,Z 500.536,A -85,B 0,C 180,E1 -22284.226,E2 -22284.226} C_VEL
LIN {X 0,Y 259.167,Z 420.078,A -85,B 0,C 180,E1 -22286.215,E2 -22286.215} C_VEL
LIN {X 0,Y 260.184,Z 406.583,A -85,B 0,C 180,E1 -22286.538,E2 -22286.538} C_VEL
LIN {X 0,Y 254.633,Z 396.157,A -85,B 0,C 180,E1 -22289.051,E2 -22289.051} C_VEL
LIN {X 0,Y 249.23,Z 386.895,A -85,B 0,C 180,E1 -22291.757,E2 -22291.757} C_VEL
LIN {X 0,Y 243.783,Z 378.413,A -85,B 0,C 180,E1 -22294.835,E2 -22294.835} C_VEL
LIN {X 0,Y 239.276,Z 371.732,A -85,B 0,C 180,E1 -22297.78,E2 -22297.78} C_VEL
LIN {X 0,Y 236.531,Z 367.843,A -85,B 0,C 180,E1 -22299.821,E2 -22299.821} C_VEL
LIN {X 0,Y 233.687,Z 363.843,A -85,B 0,C 180,E1 -22302.23,E2 -22302.23} C_VEL
LIN {X 0,Y 230.99,Z 360.249,A -85,B 0,C 180,E1 -22304.899,E2 -22304.899} C_VEL
LIN {X 0,Y 230.154,Z 358.988,A -85,B 0,C 180,E1 -22305.86,E2 -22305.86} C_VEL
LIN {X 0,Y 227.729,Z 356.09,A -85,B 0,C 180,E1 -22309.044,E2 -22309.044} C_VEL
LIN {X 0,Y 226.861,Z 354.124,A -85,B 0,C 180,E1 -22310.639,E2 -22310.639} C_VEL
LIN {X 0,Y 224.308,Z 351.267,A -85,B 0,C 180,E1 -22320,E2 -22320} C_VEL
LIN {X 0,Y 226.992,Z 354.36,A -85,B 0,C 180,E1 -22329.242,E2 -22329.242} C_VEL
LIN {X 0,Y 228.826,Z 357.745,A -85,B 0,C 180,E1 -22332.19,E2 -22332.19} C_VEL
LIN {X 0,Y 230.718,Z 359.724,A -85,B 0,C 180,E1 -22334.416,E2 -22334.416} C_VEL
LIN {X 0,Y 233.432,Z 363.614,A -85,B 0,C 180,E1 -22337.183,E2 -22337.183} C_VEL
LIN {X 0,Y 234.594,Z 365.207,A -85,B 0,C 180,E1 -22338.221,E2 -22338.221} C_VEL
LIN {X 0,Y 237.716,Z 369.513,A -85,B 0,C 180,E1 -22340.723,E2 -22340.723} C_VEL
LIN {X 0,Y 241.045,Z 374.354,A -85,B 0,C 180,E1 -22343.065,E2 -22343.065} C_VEL
LIN {X 0,Y 245.148,Z 380.425,A -85,B 0,C 180,E1 -22345.608,E2 -22345.608} C_VEL
LIN {X 0,Y 246.345,Z 382.575,A -85,B 0,C 180,E1 -22346.317,E2 -22346.317} C_VEL
LIN {X 0,Y 247.736,Z 386.802,A -85,B 0,C 180,E1 -22347.217,E2 -22347.217} C_VEL
LIN {X 0,Y 251.024,Z 401.661,A -85,B 0,C 180,E1 -22349.483,E2 -22349.483} C_VEL
LIN {X 0,Y 252.106,Z 404.559,A -85,B 0,C 180,E1 -22350.073,E2 -22350.073} C_VEL
LIN {X 0,Y 255.934,Z 413.356,A -85,B 0,C 180,E1 -22351.969,E2 -22351.969} C_VEL
LIN {X 0,Y 248.514,Z 507.819,A -85,B 0,C 180,E1 -22354.279,E2 -22354.279} C_VEL
LIN {X 0,Y 246.09,Z 524.42,A -85,B 0,C 180,E1 -22354.872,E2 -22354.872} C_VEL
LIN {X 0,Y 242.769,Z 540.177,A -85,B 0,C 180,E1 -22355.636,E2 -22355.636} C_VEL
LIN {X 0,Y 238.727,Z 555.552,A -85,B 0,C 180,E1 -22356.658,E2 -22356.658} C_VEL
LIN {X 0,Y 234.559,Z 568.727,A -85,B 0,C 180,E1 -22357.791,E2 -22357.791} C_VEL
LIN {X 0,Y 229.289,Z 582.867,A -85,B 0,C 180,E1 -22359.291,E2 -22359.291} C_VEL
LIN {X 0,Y 223.173,Z 597.324,A -85,B 0,C 180,E1 -22361.245,E2 -22361.245} C_VEL
LIN {X 0,Y 216.81,Z 610.653,A -85,B 0,C 180,E1 -22363.507,E2 -22363.507} C_VEL
LIN {X 0,Y 210.247,Z 622.852,A -85,B 0,C 180,E1 -22366.084,E2 -22366.084} C_VEL
LIN {X 0,Y 203.819,Z 634.043,A -85,B 0,C 180,E1 -22369.07,E2 -22369.07} C_VEL
LIN {X 0,Y 198.127,Z 643.662,A -85,B 0,C 180,E1 -22372.274,E2 -22372.274} C_VEL
LIN {X 0,Y 192.149,Z 653.015,A -85,B 0,C 180,E1 -22376.098,E2 -22376.098} C_VEL
LIN {X 0,Y 186.577,Z 661.697,A -85,B 0,C 180,E1 -22380.681,E2 -22380.681} C_VEL
LIN {X 0,Y 181.824,Z 669.396,A -85,B 0,C 180,E1 -22386.056,E2 -22386.056} C_VEL
LIN {X 0,Y 178.599,Z 675.271,A -85,B 0,C 180,E1 -22391.651,E2 -22391.651} C_VEL
LIN {X 0,Y 176.856,Z 678.71,A -85,B 0,C 180,E1 -22396.206,E2 -22396.206} C_VEL
LIN {X 0,Y 176.071,Z 681.222,A -85,B 0,C 180,E1 -22400.813,E2 -22400.813} C_VEL
LIN {X 0,Y 175.937,Z 682.647,A -85,B 0,C 180,E1 -22405.418,E2 -22405.418} C_VEL
LIN {X 0,Y 176.078,Z 683.184,A -85,B 0,C 180,E1 -22410,E2 -22410} C_VEL
LIN {X 0,Y 175.937,Z 682.634,A -85,B 0,C 180,E1 -22414.582,E2 -22414.582} C_VEL
LIN {X 0,Y 176.071,Z 681.195,A -85,B 0,C 180,E1 -22419.187,E2 -22419.187} C_VEL
LIN {X 0,Y 176.854,Z 678.67,A -85,B 0,C 180,E1 -22423.794,E2 -22423.794} C_VEL
LIN {X 0,Y 178.594,Z 675.217,A -85,B 0,C 180,E1 -22428.35,E2 -22428.35} C_VEL
LIN {X 0,Y 181.826,Z 669.324,A -85,B 0,C 180,E1 -22433.944,E2 -22433.944} C_VEL
LIN {X 0,Y 186.624,Z 661.598,A -85,B 0,C 180,E1 -22439.312,E2 -22439.312} C_VEL
LIN {X 0,Y 192.158,Z 652.898,A -85,B 0,C 180,E1 -22443.9,E2 -22443.9} C_VEL
LIN {X 0,Y 198.115,Z 643.52,A -85,B 0,C 180,E1 -22447.729,E2 -22447.729} C_VEL
LIN {X 0,Y 203.246,Z 634.87,A -85,B 0,C 180,E1 -22450.633,E2 -22450.633} C_VEL
LIN {X 0,Y 209.272,Z 624.381,A -85,B 0,C 180,E1 -22453.507,E2 -22453.507} C_VEL
LIN {X 0,Y 215.184,Z 613.355,A -85,B 0,C 180,E1 -22455.933,E2 -22455.933} C_VEL
LIN {X 0,Y 222.03,Z 599.393,A -85,B 0,C 180,E1 -22458.405,E2 -22458.405} C_VEL
LIN {X 0,Y 228.148,Z 585.38,A -85,B 0,C 180,E1 -22460.364,E2 -22460.364} C_VEL
LIN {X 0,Y 233.355,Z 571.751,A -85,B 0,C 180,E1 -22461.888,E2 -22461.888} C_VEL
LIN {X 0,Y 238.118,Z 557.045,A -85,B 0,C 180,E1 -22463.186,E2 -22463.186} C_VEL
LIN {X 0,Y 242.371,Z 541.088,A -85,B 0,C 180,E1 -22464.282,E2 -22464.282} C_VEL
LIN {X 0,Y 245.79,Z 524.941,A -85,B 0,C 180,E1 -22465.089,E2 -22465.089} C_VEL
LIN {X 0,Y 248.193,Z 509.198,A -85,B 0,C 180,E1 -22465.65,E2 -22465.65} C_VEL
LIN {X 0,Y 253.244,Z 445.174,A -85,B 0,C 180,E1 -22467.253,E2 -22467.253} C_VEL
LIN {X 0,Y 255.737,Z 413.163,A -85,B 0,C 180,E1 -22468.018,E2 -22468.018} C_VEL
LIN {X 0,Y 250.92,Z 402.241,A -85,B 0,C 180,E1 -22470.419,E2 -22470.419} C_VEL
LIN {X 0,Y 246.205,Z 392.489,A -85,B 0,C 180,E1 -22472.997,E2 -22472.997} C_VEL
LIN {X 0,Y 243.722,Z 387.982,A -85,B 0,C 180,E1 -22474.451,E2 -22474.451} C_VEL
LIN {X 0,Y 239.431,Z 381.28,A -85,B 0,C 180,E1 -22477.165,E2 -22477.165} C_VEL
LIN {X 0,Y 237.083,Z 377.75,A -85,B 0,C 180,E1 -22478.821,E2 -22478.821} C_VEL
LIN {X 0,Y 234.586,Z 374.12,A -85,B 0,C 180,E1 -22480.759,E2 -22480.759} C_VEL
LIN {X 0,Y 231.76,Z 370.092,A -85,B 0,C 180,E1 -22483.257,E2 -22483.257} C_VEL
LIN {X 0,Y 228.777,Z 365.774,A -85,B 0,C 180,E1 -22486.454,E2 -22486.454} C_VEL
LIN {X 0,Y 226.314,Z 362.534,A -85,B 0,C 180,E1 -22489.827,E2 -22489.827} C_VEL
LIN {X 0,Y 225.672,Z 361.052,A -85,B 0,C 180,E1 -22491.042,E2 -22491.042} C_VEL
LIN {X 0,Y 223.182,Z 357.78,A -85,B 0,C 180,E1 -22500,E2 -22500} C_VEL
LIN {X 0,Y 225.789,Z 361.269,A -85,B 0,C 180,E1 -22509.637,E2 -22509.637} C_VEL
LIN {X 0,Y 227.875,Z 364.896,A -85,B 0,C 180,E1 -22512.921,E2 -22512.921} C_VEL
LIN {X 0,Y 229.244,Z 366.315,A -85,B 0,C 180,E1 -22514.537,E2 -22514.537} C_VEL
LIN {X 0,Y 231.761,Z 370.102,A -85,B 0,C 180,E1 -22517.2,E2 -22517.2} C_VEL
LIN {X 0,Y 232.783,Z 371.47,A -85,B 0,C 180,E1 -22518.141,E2 -22518.141} C_VEL
LIN {X 0,Y 236.008,Z 376.147,A -85,B 0,C 180,E1 -22520.823,E2 -22520.823} C_VEL
LIN {X 0,Y 239.129,Z 380.876,A -85,B 0,C 180,E1 -22523.09,E2 -22523.09} C_VEL
LIN {X 0,Y 243.051,Z 386.794,A -85,B 0,C 180,E1 -22525.595,E2 -22525.595} C_VEL
LIN {X 0,Y 248.825,Z 396.441,A -85,B 0,C 180,E1 -22528.843,E2 -22528.843} C_VEL
LIN {X 0,Y 254.149,Z 406.261,A -85,B 0,C 180,E1 -22531.499,E2 -22531.499} C_VEL
LIN {X 0,Y 255.886,Z 409.595,A -85,B 0,C 180,E1 -22532.307,E2 -22532.307} C_VEL
LIN {X 0,Y 248.838,Z 500.12,A -85,B 0,C 180,E1 -22534.553,E2 -22534.553} C_VEL
LIN {X 0,Y 246.429,Z 516.904,A -85,B 0,C 180,E1 -22535.189,E2 -22535.189} C_VEL
LIN {X 0,Y 243.282,Z 532.45,A -85,B 0,C 180,E1 -22536.015,E2 -22536.015} C_VEL
LIN {X 0,Y 239.211,Z 548.405,A -85,B 0,C 180,E1 -22537.163,E2 -22537.163} C_VEL
LIN {X 0,Y 234.571,Z 563.078,A -85,B 0,C 180,E1 -22538.489,E2 -22538.489} C_VEL
LIN {X 0,Y 228.908,Z 578.235,A -85,B 0,C 180,E1 -22540.251,E2 -22540.251} C_VEL
LIN {X 0,Y 223.125,Z 591.743,A -85,B 0,C 180,E1 -22542.252,E2 -22542.252} C_VEL
LIN {X 0,Y 217.944,Z 602.472,A -85,B 0,C 180,E1 -22544.153,E2 -22544.153} C_VEL
LIN {X 0,Y 211.298,Z 615.06,A -85,B 0,C 180,E1 -22546.904,E2 -22546.904} C_VEL
LIN {X 0,Y 204.908,Z 626.174,A -85,B 0,C 180,E1 -22549.977,E2 -22549.977} C_VEL
LIN {X 0,Y 199.19,Z 635.436,A -85,B 0,C 180,E1 -22553.144,E2 -22553.144} C_VEL
LIN {X 0,Y 193.372,Z 644.445,A -85,B 0,C 180,E1 -22556.964,E2 -22556.964} C_VEL
LIN {X 0,Y 188.391,Z 651.97,A -85,B 0,C 180,E1 -22560.99,E2 -22560.99} C_VEL
LIN {X 0,Y 183.431,Z 659.518,A -85,B 0,C 180,E1 -22566.278,E2 -22566.278} C_VEL
LIN {X 0,Y 179.799,Z 665.241,A -85,B 0,C 180,E1 -22571.778,E2 -22571.778} C_VEL
LIN {X 0,Y 177.819,Z 668.584,A -85,B 0,C 180,E1 -22576.282,E2 -22576.282} C_VEL
LIN {X 0,Y 176.686,Z 671.007,A -85,B 0,C 180,E1 -22580.845,E2 -22580.845} C_VEL
LIN {X 0,Y 176.118,Z 672.506,A -85,B 0,C 180,E1 -22586.053,E2 -22586.053} C_VEL
LIN {X 0,Y 176.113,Z 672.9,A -85,B 0,C 180,E1 -22590,E2 -22590} C_VEL
LIN {X 0,Y 176.15,Z 672.41,A -85,B 0,C 180,E1 -22594.577,E2 -22594.577} C_VEL
LIN {X 0,Y 176.68,Z 671.072,A -85,B 0,C 180,E1 -22599.155,E2 -22599.155} C_VEL
LIN {X 0,Y 177.795,Z 668.68,A -85,B 0,C 180,E1 -22603.719,E2 -22603.719} C_VEL
LIN {X 0,Y 179.753,Z 665.376,A -85,B 0,C 180,E1 -22608.227,E2 -22608.227} C_VEL
LIN {X 0,Y 183.371,Z 659.692,A -85,B 0,C 180,E1 -22613.73,E2 -22613.73} C_VEL
LIN {X 0,Y 188.354,Z 652.202,A -85,B 0,C 180,E1 -22619.016,E2 -22619.016} C_VEL
LIN {X 0,Y 194.02,Z 643.636,A -85,B 0,C 180,E1 -22623.578,E2 -22623.578} C_VEL
LIN {X 0,Y 199.863,Z 634.534,A -85,B 0,C 180,E1 -22627.342,E2 -22627.342} C_VEL
LIN {X 0,Y 205.675,Z 625.083,A -85,B 0,C 180,E1 -22630.484,E2 -22630.484} C_VEL
LIN {X 0,Y 211.993,Z 614.06,A -85,B 0,C 180,E1 -22633.463,E2 -22633.463} C_VEL
LIN {X 0,Y 218.81,Z 601.006,A -85,B 0,C 180,E1 -22636.276,E2 -22636.276} C_VEL
LIN {X 0,Y 225.14,Z 587.671,A -85,B 0,C 180,E1 -22638.519,E2 -22638.519} C_VEL
LIN {X 0,Y 229.952,Z 575.939,A -85,B 0,C 180,E1 -22640.164,E2 -22640.164} C_VEL
LIN {X 0,Y 235.03,Z 562.271,A -85,B 0,C 180,E1 -22641.714,E2 -22641.714} C_VEL
LIN {X 0,Y 240.005,Z 546.445,A -85,B 0,C 180,E1 -22643.109,E2 -22643.109} C_VEL
LIN {X 0,Y 243.756,Z 531.164,A -85,B 0,C 180,E1 -22644.183,E2 -22644.183} C_VEL
LIN {X 0,Y 246.893,Z 515.084,A -85,B 0,C 180,E1 -22645.012,E2 -22645.012} C_VEL
LIN {X 0,Y 249.079,Z 499.193,A -85,B 0,C 180,E1 -22645.601,E2 -22645.601} C_VEL
LIN {X 0,Y 256.088,Z 409.806,A -85,B 0,C 180,E1 -22647.794,E2 -22647.794} C_VEL
LIN {X 0,Y 250.869,Z 399.929,A -85,B 0,C 180,E1 -22650.312,E2 -22650.312} C_VEL
LIN {X 0,Y 245.155,Z 390.059,A -85,B 0,C 180,E1 -22653.394,E2 -22653.394} C_VEL
LIN {X 0,Y 240.143,Z 382.223,A -85,B 0,C 180,E1 -22656.486,E2 -22656.486} C_VEL
LIN {X 0,Y 236.867,Z 377.31,A -85,B 0,C 180,E1 -22658.801,E2 -22658.801} C_VEL
LIN {X 0,Y 234.917,Z 374.435,A -85,B 0,C 180,E1 -22660.332,E2 -22660.332} C_VEL
LIN {X 0,Y 232.087,Z 370.403,A -85,B 0,C 180,E1 -22662.827,E2 -22662.827} C_VEL
LIN {X 0,Y 229.374,Z 366.443,A -85,B 0,C 180,E1 -22665.698,E2 -22665.698} C_VEL
LIN {X 0,Y 226.424,Z 362.596,A -85,B 0,C 180,E1 -22669.719,E2 -22669.719} C_VEL
LIN {X 0,Y 225.749,Z 361.036,A -85,B 0,C 180,E1 -22671.045,E2 -22671.045} C_VEL
LIN {X 0,Y 223.443,Z 358.318,A -85,B 0,C 180,E1 -22680,E2 -22680} C_VEL
LIN {X 0,Y 225.931,Z 361.358,A -85,B 0,C 180,E1 -22688.947,E2 -22688.947} C_VEL
LIN {X 0,Y 227.797,Z 364.76,A -85,B 0,C 180,E1 -22692.02,E2 -22692.02} C_VEL
LIN {X 0,Y 229.393,Z 366.487,A -85,B 0,C 180,E1 -22693.961,E2 -22693.961} C_VEL
LIN {X 0,Y 232.226,Z 370.554,A -85,B 0,C 180,E1 -22696.935,E2 -22696.935} C_VEL
LIN {X 0,Y 236.053,Z 376.127,A -85,B 0,C 180,E1 -22700.213,E2 -22700.213} C_VEL
LIN {X 0,Y 239.027,Z 380.549,A -85,B 0,C 180,E1 -22702.392,E2 -22702.392} C_VEL
LIN {X 0,Y 243.635,Z 387.677,A -85,B 0,C 180,E1 -22705.352,E2 -22705.352} C_VEL
LIN {X 0,Y 246.398,Z 392.687,A -85,B 0,C 180,E1 -22706.981,E2 -22706.981} C_VEL
LIN {X 0,Y 250.398,Z 400.891,A -85,B 0,C 180,E1 -22709.187,E2 -22709.187} C_VEL
LIN {X 0,Y 252.106,Z 404.559,A -85,B 0,C 180,E1 -22710.073,E2 -22710.073} C_VEL
LIN {X 0,Y 252.777,Z 407.141,A -85,B 0,C 180,E1 -22710.474,E2 -22710.474} C_VEL
LIN {X 0,Y 252.904,Z 411.539,A -85,B 0,C 180,E1 -22710.762,E2 -22710.762} C_VEL
LIN {X 0,Y 251.914,Z 419.857,A -85,B 0,C 180,E1 -22710.838,E2 -22710.838} C_VEL
LIN {X 0,Y 251.272,Z 425.529,A -85,B 0,C 180,E1 -22710.902,E2 -22710.902} C_VEL
LIN {X 0,Y 244.579,Z 507.63,A -85,B 0,C 180,E1 -22712.903,E2 -22712.903} C_VEL
LIN {X 0,Y 242.036,Z 524.474,A -85,B 0,C 180,E1 -22713.496,E2 -22713.496} C_VEL
LIN {X 0,Y 238.673,Z 540.116,A -85,B 0,C 180,E1 -22714.261,E2 -22714.261} C_VEL
LIN {X 0,Y 234.564,Z 555.351,A -85,B 0,C 180,E1 -22715.268,E2 -22715.268} C_VEL
LIN {X 0,Y 230.258,Z 568.524,A -85,B 0,C 180,E1 -22716.388,E2 -22716.388} C_VEL
LIN {X 0,Y 224.844,Z 582.663,A -85,B 0,C 180,E1 -22717.886,E2 -22717.886} C_VEL
LIN {X 0,Y 219.078,Z 595.956,A -85,B 0,C 180,E1 -22719.654,E2 -22719.654} C_VEL
LIN {X 0,Y 212.477,Z 609.427,A -85,B 0,C 180,E1 -22721.908,E2 -22721.908} C_VEL
LIN {X 0,Y 206.126,Z 620.853,A -85,B 0,C 180,E1 -22724.275,E2 -22724.275} C_VEL
LIN {X 0,Y 199.353,Z 632.34,A -85,B 0,C 180,E1 -22727.263,E2 -22727.263} C_VEL
LIN {X 0,Y 193.331,Z 642.212,A -85,B 0,C 180,E1 -22730.494,E2 -22730.494} C_VEL
LIN {X 0,Y 186.917,Z 651.707,A -85,B 0,C 180,E1 -22734.353,E2 -22734.353} C_VEL
LIN {X 0,Y 181.308,Z 659.98,A -85,B 0,C 180,E1 -22738.674,E2 -22738.674} C_VEL
LIN {X 0,Y 177.129,Z 666.309,A -85,B 0,C 180,E1 -22742.853,E2 -22742.853} C_VEL
LIN {X 0,Y 173.678,Z 671.716,A -85,B 0,C 180,E1 -22747.392,E2 -22747.392} C_VEL
LIN {X 0,Y 171.786,Z 675.062,A -85,B 0,C 180,E1 -22750.896,E2 -22750.896} C_VEL
LIN {X 0,Y 169.906,Z 678.502,A -85,B 0,C 180,E1 -22755.63,E2 -22755.63} C_VEL
LIN {X 0,Y 169.018,Z 681.013,A -85,B 0,C 180,E1 -22760.426,E2 -22760.426} C_VEL
LIN {X 0,Y 168.844,Z 682.44,A -85,B 0,C 180,E1 -22765.225,E2 -22765.225} C_VEL
LIN {X 0,Y 168.987,Z 682.977,A -85,B 0,C 180,E1 -22770,E2 -22770} C_VEL
LIN {X 0,Y 168.844,Z 682.426,A -85,B 0,C 180,E1 -22774.775,E2 -22774.775} C_VEL
LIN {X 0,Y 169.018,Z 680.985,A -85,B 0,C 180,E1 -22779.574,E2 -22779.574} C_VEL
LIN {X 0,Y 169.905,Z 678.46,A -85,B 0,C 180,E1 -22784.37,E2 -22784.37} C_VEL
LIN {X 0,Y 171.776,Z 675.006,A -85,B 0,C 180,E1 -22789.106,E2 -22789.106} C_VEL
LIN {X 0,Y 175.275,Z 669.113,A -85,B 0,C 180,E1 -22794.899,E2 -22794.899} C_VEL
LIN {X 0,Y 180.379,Z 661.386,A -85,B 0,C 180,E1 -22800.431,E2 -22800.431} C_VEL
LIN {X 0,Y 186.207,Z 652.686,A -85,B 0,C 180,E1 -22805.14,E2 -22805.14} C_VEL
LIN {X 0,Y 192.463,Z 643.308,A -85,B 0,C 180,E1 -22809.043,E2 -22809.043} C_VEL
LIN {X 0,Y 197.742,Z 634.829,A -85,B 0,C 180,E1 -22811.938,E2 -22811.938} C_VEL
LIN {X 0,Y 204.125,Z 624.169,A -85,B 0,C 180,E1 -22814.895,E2 -22814.895} C_VEL
LIN {X 0,Y 210.282,Z 613.144,A -85,B 0,C 180,E1 -22817.33,E2 -22817.33} C_VEL
LIN {X 0,Y 217.126,Z 599.647,A -85,B 0,C 180,E1 -22819.743,E2 -22819.743} C_VEL
LIN {X 0,Y 223.075,Z 586.599,A -85,B 0,C 180,E1 -22821.599,E2 -22821.599} C_VEL
LIN {X 0,Y 229.015,Z 571.537,A -85,B 0,C 180,E1 -22823.294,E2 -22823.294} C_VEL
LIN {X 0,Y 233.921,Z 556.831,A -85,B 0,C 180,E1 -22824.582,E2 -22824.582} C_VEL
LIN {X 0,Y 238.293,Z 540.872,A -85,B 0,C 180,E1 -22825.67,E2 -22825.67} C_VEL
LIN {X 0,Y 241.699,Z 525.246,A -85,B 0,C 180,E1 -22826.45,E2 -22826.45} C_VEL
LIN {X 0,Y 244.26,Z 508.977,A -85,B 0,C 180,E1 -22827.024,E2 -22827.024} C_VEL
LIN {X 0,Y 249.204,Z 448.293,A -85,B 0,C 180,E1 -22828.546,E2 -22828.546} C_VEL
LIN {X 0,Y 251.756,Z 416.052,A -85,B 0,C 180,E1 -22829.329,E2 -22829.329} C_VEL
LIN {X 0,Y 247.051,Z 405.34,A -85,B 0,C 180,E1 -22831.838,E2 -22831.838} C_VEL
LIN {X 0,Y 243.057,Z 396.938,A -85,B 0,C 180,E1 -22834.181,E2 -22834.181} C_VEL
LIN {X 0,Y 240.479,Z 392.331,A -85,B 0,C 180,E1 -22835.792,E2 -22835.792} C_VEL
LIN {X 0,Y 235.791,Z 384.847,A -85,B 0,C 180,E1 -22839.043,E2 -22839.043} C_VEL
LIN {X 0,Y 232.836,Z 380.51,A -85,B 0,C 180,E1 -22841.409,E2 -22841.409} C_VEL
LIN {X 0,Y 230.339,Z 376.795,A -85,B 0,C 180,E1 -22843.721,E2 -22843.721} C_VEL
LIN {X 0,Y 227.503,Z 372.566,A -85,B 0,C 180,E1 -22846.888,E2 -22846.888} C_VEL
LIN {X 0,Y 225.135,Z 369.246,A -85,B 0,C 180,E1 -22850.313,E2 -22850.313} C_VEL
LIN {X 0,Y 224.561,Z 367.943,A -85,B 0,C 180,E1 -22851.451,E2 -22851.451} C_VEL
LIN {X 0,Y 222.314,Z 364.848,A -85,B 0,C 180,E1 -22860,E2 -22860} C_VEL
LIN {X 0,Y 224.71,Z 368.218,A -85,B 0,C 180,E1 -22869.302,E2 -22869.302} C_VEL
LIN {X 0,Y 226.842,Z 371.919,A -85,B 0,C 180,E1 -22872.753,E2 -22872.753} C_VEL
LIN {X 0,Y 227.995,Z 373.212,A -85,B 0,C 180,E1 -22874.163,E2 -22874.163} C_VEL
LIN {X 0,Y 230.455,Z 376.924,A -85,B 0,C 180,E1 -22876.846,E2 -22876.846} C_VEL
LIN {X 0,Y 234.339,Z 382.696,A -85,B 0,C 180,E1 -22880.29,E2 -22880.29} C_VEL
LIN {X 0,Y 237.372,Z 387.452,A -85,B 0,C 180,E1 -22882.58,E2 -22882.58} C_VEL
LIN {X 0,Y 241.527,Z 394.041,A -85,B 0,C 180,E1 -22885.324,E2 -22885.324} C_VEL
LIN {X 0,Y 246.433,Z 402.499,A -85,B 0,C 180,E1 -22888.178,E2 -22888.178} C_VEL
LIN {X 0,Y 251.44,Z 412.061,A -85,B 0,C 180,E1 -22890.788,E2 -22890.788} C_VEL
LIN {X 0,Y 251.955,Z 413.03,A -85,B 0,C 180,E1 -22891.039,E2 -22891.039} C_VEL
LIN {X 0,Y 244.909,Z 500.086,A -85,B 0,C 180,E1 -22893.178,E2 -22893.178} C_VEL
LIN {X 0,Y 242.418,Z 517.123,A -85,B 0,C 180,E1 -22893.821,E2 -22893.821} C_VEL
LIN {X 0,Y 239.188,Z 532.665,A -85,B 0,C 180,E1 -22894.643,E2 -22894.643} C_VEL
LIN {X 0,Y 235.589,Z 546.64,A -85,B 0,C 180,E1 -22895.619,E2 -22895.619} C_VEL
LIN {X 0,Y 230.782,Z 561.585,A -85,B 0,C 180,E1 -22896.929,E2 -22896.929} C_VEL
LIN {X 0,Y 225.585,Z 575.424,A -85,B 0,C 180,E1 -22898.487,E2 -22898.487} C_VEL
LIN {X 0,Y 219.487,Z 589.62,A -85,B 0,C 180,E1 -22900.494,E2 -22900.494} C_VEL
LIN {X 0,Y 213.022,Z 602.684,A -85,B 0,C 180,E1 -22902.772,E2 -22902.772} C_VEL
LIN {X 0,Y 206.884,Z 613.987,A -85,B 0,C 180,E1 -22905.248,E2 -22905.248} C_VEL
LIN {X 0,Y 200.38,Z 624.911,A -85,B 0,C 180,E1 -22908.211,E2 -22908.211} C_VEL
LIN {X 0,Y 193.501,Z 635.647,A -85,B 0,C 180,E1 -22911.871,E2 -22911.871} C_VEL
LIN {X 0,Y 187.397,Z 644.657,A -85,B 0,C 180,E1 -22915.768,E2 -22915.768} C_VEL
LIN {X 0,Y 182.155,Z 652.181,A -85,B 0,C 180,E1 -22919.896,E2 -22919.896} C_VEL
LIN {X 0,Y 176.902,Z 659.728,A -85,B 0,C 180,E1 -22925.346,E2 -22925.346} C_VEL
LIN {X 0,Y 173.026,Z 665.45,A -85,B 0,C 180,E1 -22931.038,E2 -22931.038} C_VEL
LIN {X 0,Y 170.88,Z 668.793,A -85,B 0,C 180,E1 -22935.714,E2 -22935.714} C_VEL
LIN {X 0,Y 169.655,Z 671.216,A -85,B 0,C 180,E1 -22940.462,E2 -22940.462} C_VEL
LIN {X 0,Y 169.002,Z 672.819,A -85,B 0,C 180,E1 -22946.425,E2 -22946.425} C_VEL
LIN {X 0,Y 169.023,Z 673.107,A -85,B 0,C 180,E1 -22950,E2 -22950} C_VEL
LIN {X 0,Y 169.068,Z 672.617,A -85,B 0,C 180,E1 -22954.769,E2 -22954.769} C_VEL
LIN {X 0,Y 169.649,Z 671.279,A -85,B 0,C 180,E1 -22959.538,E2 -22959.538} C_VEL
LIN {X 0,Y 170.856,Z 668.889,A -85,B 0,C 180,E1 -22964.288,E2 -22964.288} C_VEL
LIN {X 0,Y 172.978,Z 665.584,A -85,B 0,C 180,E1 -22968.967,E2 -22968.967} C_VEL
LIN {X 0,Y 176.83,Z 659.901,A -85,B 0,C 180,E1 -22974.665,E2 -22974.665} C_VEL
LIN {X 0,Y 182.115,Z 652.41,A -85,B 0,C 180,E1 -22980.111,E2 -22980.111} C_VEL
LIN {X 0,Y 187.783,Z 644.265,A -85,B 0,C 180,E1 -22984.575,E2 -22984.575} C_VEL
LIN {X 0,Y 193.404,Z 635.962,A -85,B 0,C 180,E1 -22988.152,E2 -22988.152} C_VEL
LIN {X 0,Y 200.312,Z 625.288,A -85,B 0,C 180,E1 -22991.806,E2 -22991.806} C_VEL
LIN {X 0,Y 206.869,Z 614.266,A -85,B 0,C 180,E1 -22994.824,E2 -22994.824} C_VEL
LIN {X 0,Y 213.951,Z 601.211,A -85,B 0,C 180,E1 -22997.654,E2 -22997.654} C_VEL
LIN {X 0,Y 220.483,Z 587.876,A -85,B 0,C 180,E1 -22999.907,E2 -22999.907} C_VEL
LIN {X 0,Y 225.458,Z 576.142,A -85,B 0,C 180,E1 -23001.554,E2 -23001.554} C_VEL
LIN {X 0,Y 230.7,Z 562.472,A -85,B 0,C 180,E1 -23003.098,E2 -23003.098} C_VEL
LIN {X 0,Y 236.09,Z 545.625,A -85,B 0,C 180,E1 -23004.577,E2 -23004.577} C_VEL
LIN {X 0,Y 239.969,Z 530.066,A -85,B 0,C 180,E1 -23005.642,E2 -23005.642} C_VEL
LIN {X 0,Y 243.061,Z 514.365,A -85,B 0,C 180,E1 -23006.418,E2 -23006.418} C_VEL
LIN {X 0,Y 245.331,Z 497.424,A -85,B 0,C 180,E1 -23007.023,E2 -23007.023} C_VEL
LIN {X 0,Y 252.137,Z 413.2,A -85,B 0,C 180,E1 -23009.074,E2 -23009.074} C_VEL
LIN {X 0,Y 247.372,Z 404.085,A -85,B 0,C 180,E1 -23011.525,E2 -23011.525} C_VEL
LIN {X 0,Y 242.617,Z 395.706,A -85,B 0,C 180,E1 -23014.245,E2 -23014.245} C_VEL
LIN {X 0,Y 238.235,Z 388.591,A -85,B 0,C 180,E1 -23017.082,E2 -23017.082} C_VEL
LIN {X 0,Y 234.856,Z 383.369,A -85,B 0,C 180,E1 -23019.585,E2 -23019.585} C_VEL
LIN {X 0,Y 232.952,Z 380.551,A -85,B 0,C 180,E1 -23021.161,E2 -23021.161} C_VEL
LIN {X 0,Y 230.557,Z 376.971,A -85,B 0,C 180,E1 -23023.395,E2 -23023.395} C_VEL
LIN {X 0,Y 227.697,Z 372.675,A -85,B 0,C 180,E1 -23026.615,E2 -23026.615} C_VEL
LIN {X 0,Y 225.445,Z 369.75,A -85,B 0,C 180,E1 -23029.844,E2 -23029.844} C_VEL
LIN {X 0,Y 224.647,Z 367.957,A -85,B 0,C 180,E1 -23031.454,E2 -23031.454} C_VEL
LIN {X 0,Y 222.577,Z 365.372,A -85,B 0,C 180,E1 -23040,E2 -23040} C_VEL
LIN {X 0,Y 224.828,Z 368.2,A -85,B 0,C 180,E1 -23048.539,E2 -23048.539} C_VEL
LIN {X 0,Y 226.611,Z 371.593,A -85,B 0,C 180,E1 -23051.63,E2 -23051.63} C_VEL
LIN {X 0,Y 228.149,Z 373.362,A -85,B 0,C 180,E1 -23053.584,E2 -23053.584} C_VEL
LIN {X 0,Y 231.444,Z 378.327,A -85,B 0,C 180,E1 -23057.107,E2 -23057.107} C_VEL
LIN {X 0,Y 234.443,Z 382.765,A -85,B 0,C 180,E1 -23059.72,E2 -23059.72} C_VEL
LIN {X 0,Y 237.21,Z 386.997,A -85,B 0,C 180,E1 -23061.828,E2 -23061.828} C_VEL
LIN {X 0,Y 241.549,Z 393.975,A -85,B 0,C 180,E1 -23064.735,E2 -23064.735} C_VEL
LIN {X 0,Y 244.032,Z 398.677,A -85,B 0,C 180,E1 -23066.267,E2 -23066.267} C_VEL
LIN {X 0,Y 248.219,Z 407.625,A -85,B 0,C 180,E1 -23068.678,E2 -23068.678} C_VEL
LIN {X 0,Y 252,Z 416.389,A -85,B 0,C 180,E1 -23070.682,E2 -23070.682} C_VEL
LIN {X 0,Y 251.272,Z 425.529,A -85,B 0,C 180,E1 -23070.902,E2 -23070.902} C_VEL
LIN {X 0,Y 250.504,Z 431.38,A -85,B 0,C 180,E1 -23070.929,E2 -23070.929} C_VEL
LIN {X 0,Y 245.916,Z 450.459,A -85,B 0,C 180,E1 -23070.206,E2 -23070.206} C_VEL
LIN {X 0,Y 245.083,Z 456.319,A -85,B 0,C 180,E1 -23070.207,E2 -23070.207} C_VEL
LIN {X 0,Y 240.641,Z 508.862,A -85,B 0,C 180,E1 -23071.528,E2 -23071.528} C_VEL
LIN {X 0,Y 237.858,Z 526.253,A -85,B 0,C 180,E1 -23072.158,E2 -23072.158} C_VEL
LIN {X 0,Y 234.057,Z 542.636,A -85,B 0,C 180,E1 -23072.979,E2 -23072.979} C_VEL
LIN {X 0,Y 229.884,Z 557.139,A -85,B 0,C 180,E1 -23073.978,E2 -23073.978} C_VEL
LIN {X 0,Y 225.49,Z 570.092,A -85,B 0,C 180,E1 -23075.101,E2 -23075.101} C_VEL
LIN {X 0,Y 219.324,Z 585.321,A -85,B 0,C 180,E1 -23076.766,E2 -23076.766} C_VEL
LIN {X 0,Y 212.878,Z 599.199,A -85,B 0,C 180,E1 -23078.716,E2 -23078.716} C_VEL
LIN {X 0,Y 206.66,Z 611.221,A -85,B 0,C 180,E1 -23080.829,E2 -23080.829} C_VEL
LIN {X 0,Y 200.152,Z 622.438,A -85,B 0,C 180,E1 -23083.231,E2 -23083.231} C_VEL
LIN {X 0,Y 193.18,Z 633.628,A -85,B 0,C 180,E1 -23086.273,E2 -23086.273} C_VEL
LIN {X 0,Y 186.083,Z 644.487,A -85,B 0,C 180,E1 -23090.055,E2 -23090.055} C_VEL
LIN {X 0,Y 179.603,Z 653.615,A -85,B 0,C 180,E1 -23094.059,E2 -23094.059} C_VEL
LIN {X 0,Y 174.15,Z 661.279,A -85,B 0,C 180,E1 -23098.357,E2 -23098.357} C_VEL
LIN {X 0,Y 168.755,Z 668.978,A -85,B 0,C 180,E1 -23104.07,E2 -23104.07} C_VEL
LIN {X 0,Y 164.992,Z 674.853,A -85,B 0,C 180,E1 -23110.077,E2 -23110.077} C_VEL
LIN {X 0,Y 162.978,Z 678.293,A -85,B 0,C 180,E1 -23115.005,E2 -23115.005} C_VEL
LIN {X 0,Y 161.954,Z 680.805,A -85,B 0,C 180,E1 -23120.004,E2 -23120.004} C_VEL
LIN {X 0,Y 161.735,Z 682.232,A -85,B 0,C 180,E1 -23125.014,E2 -23125.014} C_VEL
LIN {X 0,Y 161.898,Z 682.77,A -85,B 0,C 180,E1 -23130,E2 -23130} C_VEL
LIN {X 0,Y 161.735,Z 682.217,A -85,B 0,C 180,E1 -23134.986,E2 -23134.986} C_VEL
LIN {X 0,Y 161.954,Z 680.776,A -85,B 0,C 180,E1 -23139.996,E2 -23139.996} C_VEL
LIN {X 0,Y 162.976,Z 678.251,A -85,B 0,C 180,E1 -23144.995,E2 -23144.995} C_VEL
LIN {X 0,Y 165.434,Z 673.985,A -85,B 0,C 180,E1 -23150.836,E2 -23150.836} C_VEL
LIN {X 0,Y 168.759,Z 668.901,A -85,B 0,C 180,E1 -23155.93,E2 -23155.93} C_VEL
LIN {X 0,Y 174.202,Z 661.174,A -85,B 0,C 180,E1 -23161.632,E2 -23161.632} C_VEL
LIN {X 0,Y 180.357,Z 652.473,A -85,B 0,C 180,E1 -23166.459,E2 -23166.459} C_VEL
LIN {X 0,Y 186.896,Z 643.094,A -85,B 0,C 180,E1 -23170.441,E2 -23170.441} C_VEL
LIN {X 0,Y 193.193,Z 633.446,A -85,B 0,C 180,E1 -23173.724,E2 -23173.724} C_VEL
LIN {X 0,Y 200.132,Z 622.213,A -85,B 0,C 180,E1 -23176.775,E2 -23176.775} C_VEL
LIN {X 0,Y 207.156,Z 609.991,A -85,B 0,C 180,E1 -23179.384,E2 -23179.384} C_VEL
LIN {X 0,Y 213.453,Z 597.661,A -85,B 0,C 180,E1 -23181.488,E2 -23181.488} C_VEL
LIN {X 0,Y 219.918,Z 583.523,A -85,B 0,C 180,E1 -23183.41,E2 -23183.41} C_VEL
LIN {X 0,Y 225.449,Z 569.629,A -85,B 0,C 180,E1 -23184.914,E2 -23184.914} C_VEL
LIN {X 0,Y 230.8,Z 553.616,A -85,B 0,C 180,E1 -23186.271,E2 -23186.271} C_VEL
LIN {X 0,Y 235.225,Z 537.182,A -85,B 0,C 180,E1 -23187.305,E2 -23187.305} C_VEL
LIN {X 0,Y 238.65,Z 520.717,A -85,B 0,C 180,E1 -23188.035,E2 -23188.035} C_VEL
LIN {X 0,Y 240.852,Z 504.809,A -85,B 0,C 180,E1 -23188.564,E2 -23188.564} C_VEL
LIN {X 0,Y 247.951,Z 419.317,A -85,B 0,C 180,E1 -23190.642,E2 -23190.642} C_VEL
LIN {X 0,Y 244.233,Z 410.537,A -85,B 0,C 180,E1 -23192.761,E2 -23192.761} C_VEL
LIN {X 0,Y 239.955,Z 401.206,A -85,B 0,C 180,E1 -23195.44,E2 -23195.44} C_VEL
LIN {X 0,Y 235.633,Z 393.97,A -85,B 0,C 180,E1 -23198.398,E2 -23198.398} C_VEL
LIN {X 0,Y 233.184,Z 390.071,A -85,B 0,C 180,E1 -23200.295,E2 -23200.295} C_VEL
LIN {X 0,Y 231.234,Z 387.065,A -85,B 0,C 180,E1 -23201.963,E2 -23201.963} C_VEL
LIN {X 0,Y 228.725,Z 383.207,A -85,B 0,C 180,E1 -23204.404,E2 -23204.404} C_VEL
LIN {X 0,Y 226.328,Z 379.451,A -85,B 0,C 180,E1 -23207.218,E2 -23207.218} C_VEL
LIN {X 0,Y 223.997,Z 376.045,A -85,B 0,C 180,E1 -23210.747,E2 -23210.747} C_VEL
LIN {X 0,Y 223.461,Z 374.844,A -85,B 0,C 180,E1 -23211.864,E2 -23211.864} C_VEL
LIN {X 0,Y 221.446,Z 371.918,A -85,B 0,C 180,E1 -23220,E2 -23220} C_VEL
LIN {X 0,Y 223.626,Z 375.1,A -85,B 0,C 180,E1 -23228.927,E2 -23228.927} C_VEL
LIN {X 0,Y 225.648,Z 378.75,A -85,B 0,C 180,E1 -23232.365,E2 -23232.365} C_VEL
LIN {X 0,Y 226.776,Z 380.151,A -85,B 0,C 180,E1 -23233.812,E2 -23233.812} C_VEL
LIN {X 0,Y 229.999,Z 385.125,A -85,B 0,C 180,E1 -23237.336,E2 -23237.336} C_VEL
LIN {X 0,Y 232.875,Z 389.572,A -85,B 0,C 180,E1 -23239.905,E2 -23239.905} C_VEL
LIN {X 0,Y 236.751,Z 395.75,A -85,B 0,C 180,E1 -23242.862,E2 -23242.862} C_VEL
LIN {X 0,Y 241.449,Z 403.781,A -85,B 0,C 180,E1 -23245.946,E2 -23245.946} C_VEL
LIN {X 0,Y 246.496,Z 413.186,A -85,B 0,C 180,E1 -23248.849,E2 -23248.849} C_VEL
LIN {X 0,Y 248.115,Z 416.483,A -85,B 0,C 180,E1 -23249.717,E2 -23249.717} C_VEL
LIN {X 0,Y 241.116,Z 500.234,A -85,B 0,C 180,E1 -23251.768,E2 -23251.768} C_VEL
LIN {X 0,Y 238.71,Z 516.427,A -85,B 0,C 180,E1 -23252.371,E2 -23252.371} C_VEL
LIN {X 0,Y 235.232,Z 532.88,A -85,B 0,C 180,E1 -23253.223,E2 -23253.223} C_VEL
LIN {X 0,Y 230.903,Z 548.833,A -85,B 0,C 180,E1 -23254.351,E2 -23254.351} C_VEL
LIN {X 0,Y 225.996,Z 563.504,A -85,B 0,C 180,E1 -23255.666,E2 -23255.666} C_VEL
LIN {X 0,Y 219.923,Z 578.779,A -85,B 0,C 180,E1 -23257.433,E2 -23257.433} C_VEL
LIN {X 0,Y 213.255,Z 593.334,A -85,B 0,C 180,E1 -23259.616,E2 -23259.616} C_VEL
LIN {X 0,Y 207.192,Z 604.834,A -85,B 0,C 180,E1 -23261.734,E2 -23261.734} C_VEL
LIN {X 0,Y 200.198,Z 616.927,A -85,B 0,C 180,E1 -23264.497,E2 -23264.497} C_VEL
LIN {X 0,Y 193.26,Z 628.041,A -85,B 0,C 180,E1 -23267.72,E2 -23267.72} C_VEL
LIN {X 0,Y 186.237,Z 638.3,A -85,B 0,C 180,E1 -23271.49,E2 -23271.49} C_VEL
LIN {X 0,Y 180.089,Z 646.861,A -85,B 0,C 180,E1 -23275.538,E2 -23275.538} C_VEL
LIN {X 0,Y 174.764,Z 654.018,A -85,B 0,C 180,E1 -23279.823,E2 -23279.823} C_VEL
LIN {X 0,Y 170.412,Z 659.938,A -85,B 0,C 180,E1 -23284.34,E2 -23284.34} C_VEL
LIN {X 0,Y 166.284,Z 665.66,A -85,B 0,C 180,E1 -23290.238,E2 -23290.238} C_VEL
LIN {X 0,Y 163.969,Z 669.002,A -85,B 0,C 180,E1 -23295.098,E2 -23295.098} C_VEL
LIN {X 0,Y 162.648,Z 671.424,A -85,B 0,C 180,E1 -23300.047,E2 -23300.047} C_VEL
LIN {X 0,Y 162.002,Z 672.792,A -85,B 0,C 180,E1 -23305.022,E2 -23305.022} C_VEL
LIN {X 0,Y 161.936,Z 673.314,A -85,B 0,C 180,E1 -23310,E2 -23310} C_VEL
LIN {X 0,Y 162.002,Z 672.824,A -85,B 0,C 180,E1 -23314.977,E2 -23314.977} C_VEL
LIN {X 0,Y 162.642,Z 671.487,A -85,B 0,C 180,E1 -23319.953,E2 -23319.953} C_VEL
LIN {X 0,Y 163.945,Z 669.096,A -85,B 0,C 180,E1 -23324.904,E2 -23324.904} C_VEL
LIN {X 0,Y 166.232,Z 665.792,A -85,B 0,C 180,E1 -23329.769,E2 -23329.769} C_VEL
LIN {X 0,Y 170.352,Z 660.108,A -85,B 0,C 180,E1 -23335.669,E2 -23335.669} C_VEL
LIN {X 0,Y 175.948,Z 652.618,A -85,B 0,C 180,E1 -23341.283,E2 -23341.283} C_VEL
LIN {X 0,Y 181.58,Z 644.92,A -85,B 0,C 180,E1 -23345.629,E2 -23345.629} C_VEL
LIN {X 0,Y 187.831,Z 636.169,A -85,B 0,C 180,E1 -23349.5,E2 -23349.5} C_VEL
LIN {X 0,Y 195.056,Z 625.494,A -85,B 0,C 180,E1 -23353.202,E2 -23353.202} C_VEL
LIN {X 0,Y 201.868,Z 614.471,A -85,B 0,C 180,E1 -23356.252,E2 -23356.252} C_VEL
LIN {X 0,Y 209.217,Z 601.415,A -85,B 0,C 180,E1 -23359.096,E2 -23359.096} C_VEL
LIN {X 0,Y 215.96,Z 588.08,A -85,B 0,C 180,E1 -23361.354,E2 -23361.354} C_VEL
LIN {X 0,Y 221.111,Z 576.345,A -85,B 0,C 180,E1 -23362.995,E2 -23362.995} C_VEL
LIN {X 0,Y 226.494,Z 562.675,A -85,B 0,C 180,E1 -23364.54,E2 -23364.54} C_VEL
LIN {X 0,Y 232.035,Z 545.825,A -85,B 0,C 180,E1 -23366.01,E2 -23366.01} C_VEL
LIN {X 0,Y 236.046,Z 530.264,A -85,B 0,C 180,E1 -23367.06,E2 -23367.06} C_VEL
LIN {X 0,Y 239.22,Z 514.559,A -85,B 0,C 180,E1 -23367.83,E2 -23367.83} C_VEL
LIN {X 0,Y 241.527,Z 497.819,A -85,B 0,C 180,E1 -23368.427,E2 -23368.427} C_VEL
LIN {X 0,Y 248.258,Z 416.571,A -85,B 0,C 180,E1 -23370.419,E2 -23370.419} C_VEL
LIN {X 0,Y 243.534,Z 407.399,A -85,B 0,C 180,E1 -23373.039,E2 -23373.039} C_VEL
LIN {X 0,Y 238.785,Z 398.962,A -85,B 0,C 180,E1 -23376.001,E2 -23376.001} C_VEL
LIN {X 0,Y 234.168,Z 391.345,A -85,B 0,C 180,E1 -23379.35,E2 -23379.35} C_VEL
LIN {X 0,Y 231.449,Z 387.21,A -85,B 0,C 180,E1 -23381.637,E2 -23381.637} C_VEL
LIN {X 0,Y 229.047,Z 383.573,A -85,B 0,C 180,E1 -23383.969,E2 -23383.969} C_VEL
LIN {X 0,Y 226.482,Z 379.529,A -85,B 0,C 180,E1 -23386.998,E2 -23386.998} C_VEL
LIN {X 0,Y 224.235,Z 376.391,A -85,B 0,C 180,E1 -23390.415,E2 -23390.415} C_VEL
LIN {X 0,Y 223.557,Z 374.881,A -85,B 0,C 180,E1 -23391.867,E2 -23391.867} C_VEL
LIN {X 0,Y 221.71,Z 372.427,A -85,B 0,C 180,E1 -23400,E2 -23400} C_VEL
LIN {X 0,Y 223.782,Z 375.191,A -85,B 0,C 180,E1 -23408.238,E2 -23408.238} C_VEL
LIN {X 0,Y 225.551,Z 378.549,A -85,B 0,C 180,E1 -23411.4,E2 -23411.4} C_VEL
LIN {X 0,Y 226.872,Z 380.177,A -85,B 0,C 180,E1 -23413.149,E2 -23413.149} C_VEL
LIN {X 0,Y 229.977,Z 384.987,A -85,B 0,C 180,E1 -23416.612,E2 -23416.612} C_VEL
LIN {X 0,Y 233.035,Z 389.681,A -85,B 0,C 180,E1 -23419.374,E2 -23419.374} C_VEL
LIN {X 0,Y 236.691,Z 395.501,A -85,B 0,C 180,E1 -23422.189,E2 -23422.189} C_VEL
LIN {X 0,Y 240.456,Z 402.004,A -85,B 0,C 180,E1 -23424.732,E2 -23424.732} C_VEL
LIN {X 0,Y 244.844,Z 411.547,A -85,B 0,C 180,E1 -23427.455,E2 -23427.455} C_VEL
LIN {X 0,Y 248.135,Z 419.502,A -85,B 0,C 180,E1 -23429.334,E2 -23429.334} C_VEL
LIN {X 0,Y 245.083,Z 456.319,A -85,B 0,C 180,E1 -23430.207,E2 -23430.207} C_VEL
LIN {X 0,Y 244.264,Z 462.176,A -85,B 0,C 180,E1 -23430.213,E2 -23430.213} C_VEL
LIN {X 0,Y 239.761,Z 481.27,A -85,B 0,C 180,E1 -23429.478,E2 -23429.478} C_VEL
LIN {X 0,Y 238.948,Z 487.126,A -85,B 0,C 180,E1 -23429.484,E2 -23429.484} C_VEL
LIN {X 0,Y 236.782,Z 510.141,A -85,B 0,C 180,E1 -23430.108,E2 -23430.108} C_VEL
LIN {X 0,Y 233.925,Z 527.126,A -85,B 0,C 180,E1 -23430.727,E2 -23430.727} C_VEL
LIN {X 0,Y 229.937,Z 543.739,A -85,B 0,C 180,E1 -23431.571,E2 -23431.571} C_VEL
LIN {X 0,Y 225.314,Z 558.927,A -85,B 0,C 180,E1 -23432.63,E2 -23432.63} C_VEL
LIN {X 0,Y 220.187,Z 573.122,A -85,B 0,C 180,E1 -23433.915,E2 -23433.915} C_VEL
LIN {X 0,Y 214.504,Z 586.544,A -85,B 0,C 180,E1 -23435.413,E2 -23435.413} C_VEL
LIN {X 0,Y 207.667,Z 600.582,A -85,B 0,C 180,E1 -23437.427,E2 -23437.427} C_VEL
LIN {X 0,Y 200.887,Z 612.974,A -85,B 0,C 180,E1 -23439.677,E2 -23439.677} C_VEL
LIN {X 0,Y 194.236,Z 623.955,A -85,B 0,C 180,E1 -23442.12,E2 -23442.12} C_VEL
LIN {X 0,Y 186.194,Z 636.221,A -85,B 0,C 180,E1 -23445.635,E2 -23445.635} C_VEL
LIN {X 0,Y 179.731,Z 645.52,A -85,B 0,C 180,E1 -23449.083,E2 -23449.083} C_VEL
LIN {X 0,Y 173.059,Z 654.424,A -85,B 0,C 180,E1 -23453.202,E2 -23453.202} C_VEL
LIN {X 0,Y 168.051,Z 661.069,A -85,B 0,C 180,E1 -23457.067,E2 -23457.067} C_VEL
LIN {X 0,Y 162.292,Z 668.768,A -85,B 0,C 180,E1 -23462.955,E2 -23462.955} C_VEL
LIN {X 0,Y 158.238,Z 674.643,A -85,B 0,C 180,E1 -23469.188,E2 -23469.188} C_VEL
LIN {X 0,Y 156.045,Z 678.084,A -85,B 0,C 180,E1 -23474.322,E2 -23474.322} C_VEL
LIN {X 0,Y 154.911,Z 680.596,A -85,B 0,C 180,E1 -23479.545,E2 -23479.545} C_VEL
LIN {X 0,Y 154.635,Z 682.024,A -85,B 0,C 180,E1 -23484.785,E2 -23484.785} C_VEL
LIN {X 0,Y 154.797,Z 682.563,A -85,B 0,C 180,E1 -23490,E2 -23490} C_VEL
LIN {X 0,Y 154.635,Z 682.009,A -85,B 0,C 180,E1 -23495.215,E2 -23495.215} C_VEL
LIN {X 0,Y 154.911,Z 680.566,A -85,B 0,C 180,E1 -23500.456,E2 -23500.456} C_VEL
LIN {X 0,Y 156.043,Z 678.04,A -85,B 0,C 180,E1 -23505.678,E2 -23505.678} C_VEL
LIN {X 0,Y 158.536,Z 674.067,A -85,B 0,C 180,E1 -23511.419,E2 -23511.419} C_VEL
LIN {X 0,Y 162.297,Z 668.689,A -85,B 0,C 180,E1 -23517.044,E2 -23517.044} C_VEL
LIN {X 0,Y 168.104,Z 660.962,A -85,B 0,C 180,E1 -23522.922,E2 -23522.922} C_VEL
LIN {X 0,Y 174.633,Z 652.262,A -85,B 0,C 180,E1 -23527.859,E2 -23527.859} C_VEL
LIN {X 0,Y 181.444,Z 642.881,A -85,B 0,C 180,E1 -23531.924,E2 -23531.924} C_VEL
LIN {X 0,Y 188.058,Z 633.233,A -85,B 0,C 180,E1 -23535.239,E2 -23535.239} C_VEL
LIN {X 0,Y 195.287,Z 622.001,A -85,B 0,C 180,E1 -23538.309,E2 -23538.309} C_VEL
LIN {X 0,Y 202.568,Z 609.779,A -85,B 0,C 180,E1 -23540.921,E2 -23540.921} C_VEL
LIN {X 0,Y 209.576,Z 596.536,A -85,B 0,C 180,E1 -23543.15,E2 -23543.15} C_VEL
LIN {X 0,Y 215.747,Z 583.311,A -85,B 0,C 180,E1 -23544.93,E2 -23544.93} C_VEL
LIN {X 0,Y 221.424,Z 569.415,A -85,B 0,C 180,E1 -23546.426,E2 -23546.426} C_VEL
LIN {X 0,Y 226.914,Z 553.401,A -85,B 0,C 180,E1 -23547.771,E2 -23547.771} C_VEL
LIN {X 0,Y 231.346,Z 537.412,A -85,B 0,C 180,E1 -23548.762,E2 -23548.762} C_VEL
LIN {X 0,Y 234.842,Z 521.166,A -85,B 0,C 180,E1 -23549.48,E2 -23549.48} C_VEL
LIN {X 0,Y 237.272,Z 503.94,A -85,B 0,C 180,E1 -23550.054,E2 -23550.054} C_VEL
LIN {X 0,Y 244.239,Z 422.415,A -85,B 0,C 180,E1 -23552.025,E2 -23552.025} C_VEL
LIN {X 0,Y 239.835,Z 411.891,A -85,B 0,C 180,E1 -23554.763,E2 -23554.763} C_VEL
LIN {X 0,Y 237.076,Z 406.028,A -85,B 0,C 180,E1 -23556.632,E2 -23556.632} C_VEL
LIN {X 0,Y 233.214,Z 399.35,A -85,B 0,C 180,E1 -23559.47,E2 -23559.47} C_VEL
LIN {X 0,Y 229.771,Z 393.765,A -85,B 0,C 180,E1 -23562.42,E2 -23562.42} C_VEL
LIN {X 0,Y 227.34,Z 389.921,A -85,B 0,C 180,E1 -23564.881,E2 -23564.881} C_VEL
LIN {X 0,Y 225.022,Z 386.177,A -85,B 0,C 180,E1 -23567.733,E2 -23567.733} C_VEL
LIN {X 0,Y 222.831,Z 382.755,A -85,B 0,C 180,E1 -23571.27,E2 -23571.27} C_VEL
LIN {X 0,Y 222.372,Z 381.754,A -85,B 0,C 180,E1 -23572.281,E2 -23572.281} C_VEL
LIN {X 0,Y 220.577,Z 378.994,A -85,B 0,C 180,E1 -23580,E2 -23580} C_VEL
LIN {X 0,Y 222.582,Z 382.087,A -85,B 0,C 180,E1 -23588.626,E2 -23588.626} C_VEL
LIN {X 0,Y 224.785,Z 385.946,A -85,B 0,C 180,E1 -23592.413,E2 -23592.413} C_VEL
LIN {X 0,Y 225.53,Z 386.972,A -85,B 0,C 180,E1 -23593.401,E2 -23593.401} C_VEL
LIN {X 0,Y 228.449,Z 391.66,A -85,B 0,C 180,E1 -23596.747,E2 -23596.747} C_VEL
LIN {X 0,Y 231.305,Z 396.201,A -85,B 0,C 180,E1 -23599.41,E2 -23599.41} C_VEL
LIN {X 0,Y 235.356,Z 403.022,A -85,B 0,C 180,E1 -23602.611,E2 -23602.611} C_VEL
LIN {X 0,Y 239.787,Z 410.855,A -85,B 0,C 180,E1 -23605.598,E2 -23605.598} C_VEL
LIN {X 0,Y 244.366,Z 419.861,A -85,B 0,C 180,E1 -23608.331,E2 -23608.331} C_VEL
LIN {X 0,Y 237.451,Z 500.559,A -85,B 0,C 180,E1 -23610.317,E2 -23610.317} C_VEL
LIN {X 0,Y 234.831,Z 517.56,A -85,B 0,C 180,E1 -23610.95,E2 -23610.95} C_VEL
LIN {X 0,Y 231.423,Z 533.096,A -85,B 0,C 180,E1 -23611.754,E2 -23611.754} C_VEL
LIN {X 0,Y 226.979,Z 549.047,A -85,B 0,C 180,E1 -23612.874,E2 -23612.874} C_VEL
LIN {X 0,Y 221.921,Z 563.717,A -85,B 0,C 180,E1 -23614.173,E2 -23614.173} C_VEL
LIN {X 0,Y 215.933,Z 578.407,A -85,B 0,C 180,E1 -23615.863,E2 -23615.863} C_VEL
LIN {X 0,Y 209.353,Z 592.379,A -85,B 0,C 180,E1 -23617.918,E2 -23617.918} C_VEL
LIN {X 0,Y 203.578,Z 603.108,A -85,B 0,C 180,E1 -23619.815,E2 -23619.815} C_VEL
LIN {X 0,Y 197.118,Z 614.234,A -85,B 0,C 180,E1 -23622.285,E2 -23622.285} C_VEL
LIN {X 0,Y 189.984,Z 625.333,A -85,B 0,C 180,E1 -23625.344,E2 -23625.344} C_VEL
LIN {X 0,Y 182.47,Z 636.069,A -85,B 0,C 180,E1 -23629.098,E2 -23629.098} C_VEL
LIN {X 0,Y 175.736,Z 645.078,A -85,B 0,C 180,E1 -23633.139,E2 -23633.139} C_VEL
LIN {X 0,Y 169.904,Z 652.603,A -85,B 0,C 180,E1 -23637.47,E2 -23637.47} C_VEL
LIN {X 0,Y 163.968,Z 660.149,A -85,B 0,C 180,E1 -23643.253,E2 -23643.253} C_VEL
LIN {X 0,Y 159.575,Z 665.869,A -85,B 0,C 180,E1 -23649.37,E2 -23649.37} C_VEL
LIN {X 0,Y 157.061,Z 669.212,A -85,B 0,C 180,E1 -23654.426,E2 -23654.426} C_VEL
LIN {X 0,Y 155.632,Z 671.632,A -85,B 0,C 180,E1 -23659.593,E2 -23659.593} C_VEL
LIN {X 0,Y 154.93,Z 673,A -85,B 0,C 180,E1 -23664.795,E2 -23664.795} C_VEL
LIN {X 0,Y 154.853,Z 673.521,A -85,B 0,C 180,E1 -23670,E2 -23670} C_VEL
LIN {X 0,Y 154.93,Z 673.031,A -85,B 0,C 180,E1 -23675.205,E2 -23675.205} C_VEL
LIN {X 0,Y 155.626,Z 671.694,A -85,B 0,C 180,E1 -23680.407,E2 -23680.407} C_VEL
LIN {X 0,Y 157.036,Z 669.305,A -85,B 0,C 180,E1 -23685.576,E2 -23685.576} C_VEL
LIN {X 0,Y 159.503,Z 666,A -85,B 0,C 180,E1 -23690.64,E2 -23690.64} C_VEL
LIN {X 0,Y 163.931,Z 660.316,A -85,B 0,C 180,E1 -23696.753,E2 -23696.753} C_VEL
LIN {X 0,Y 169.861,Z 652.826,A -85,B 0,C 180,E1 -23702.539,E2 -23702.539} C_VEL
LIN {X 0,Y 176.45,Z 644.333,A -85,B 0,C 180,E1 -23707.402,E2 -23707.402} C_VEL
LIN {X 0,Y 183.278,Z 635.154,A -85,B 0,C 180,E1 -23711.412,E2 -23711.412} C_VEL
LIN {X 0,Y 189.915,Z 625.7,A -85,B 0,C 180,E1 -23714.677,E2 -23714.677} C_VEL
LIN {X 0,Y 195.941,Z 616.369,A -85,B 0,C 180,E1 -23717.331,E2 -23717.331} C_VEL
LIN {X 0,Y 202.382,Z 605.529,A -85,B 0,C 180,E1 -23719.816,E2 -23719.816} C_VEL
LIN {X 0,Y 209.273,Z 592.954,A -85,B 0,C 180,E1 -23722.11,E2 -23722.11} C_VEL
LIN {X 0,Y 215.633,Z 579.494,A -85,B 0,C 180,E1 -23724.134,E2 -23724.134} C_VEL
LIN {X 0,Y 221.838,Z 564.493,A -85,B 0,C 180,E1 -23725.858,E2 -23725.858} C_VEL
LIN {X 0,Y 226.903,Z 550.018,A -85,B 0,C 180,E1 -23727.156,E2 -23727.156} C_VEL
LIN {X 0,Y 231.301,Z 534.355,A -85,B 0,C 180,E1 -23728.295,E2 -23728.295} C_VEL
LIN {X 0,Y 234.657,Z 519.496,A -85,B 0,C 180,E1 -23729.099,E2 -23729.099} C_VEL
LIN {X 0,Y 237.457,Z 501.974,A -85,B 0,C 180,E1 -23729.768,E2 -23729.768} C_VEL
LIN {X 0,Y 241.455,Z 456.683,A -85,B 0,C 180,E1 -23730.907,E2 -23730.907} C_VEL
LIN {X 0,Y 244.609,Z 420.076,A -85,B 0,C 180,E1 -23731.758,E2 -23731.758} C_VEL
LIN {X 0,Y 239.587,Z 410.329,A -85,B 0,C 180,E1 -23734.77,E2 -23734.77} C_VEL
LIN {X 0,Y 235.116,Z 402.355,A -85,B 0,C 180,E1 -23737.843,E2 -23737.843} C_VEL
LIN {X 0,Y 231.507,Z 396.375,A -85,B 0,C 180,E1 -23740.723,E2 -23740.723} C_VEL
LIN {X 0,Y 229.178,Z 392.736,A -85,B 0,C 180,E1 -23742.861,E2 -23742.861} C_VEL
LIN {X 0,Y 227.613,Z 390.213,A -85,B 0,C 180,E1 -23744.497,E2 -23744.497} C_VEL
LIN {X 0,Y 225.155,Z 386.249,A -85,B 0,C 180,E1 -23747.547,E2 -23747.547} C_VEL
LIN {X 0,Y 223.074,Z 383.096,A -85,B 0,C 180,E1 -23750.936,E2 -23750.936} C_VEL
LIN {X 0,Y 222.586,Z 381.879,A -85,B 0,C 180,E1 -23752.06,E2 -23752.06} C_VEL
LIN {X 0,Y 220.845,Z 379.477,A -85,B 0,C 180,E1 -23760,E2 -23760} C_VEL
LIN {X 0,Y 222.744,Z 382.17,A -85,B 0,C 180,E1 -23767.934,E2 -23767.934} C_VEL
LIN {X 0,Y 224.419,Z 385.42,A -85,B 0,C 180,E1 -23771.058,E2 -23771.058} C_VEL
LIN {X 0,Y 225.611,Z 386.964,A -85,B 0,C 180,E1 -23772.709,E2 -23772.709} C_VEL
LIN {X 0,Y 228.488,Z 391.595,A -85,B 0,C 180,E1 -23776.071,E2 -23776.071} C_VEL
LIN {X 0,Y 231.405,Z 396.231,A -85,B 0,C 180,E1 -23778.825,E2 -23778.825} C_VEL
LIN {X 0,Y 234.84,Z 401.904,A -85,B 0,C 180,E1 -23781.588,E2 -23781.588} C_VEL
LIN {X 0,Y 238.231,Z 408.065,A -85,B 0,C 180,E1 -23783.994,E2 -23783.994} C_VEL
LIN {X 0,Y 242.542,Z 417.855,A -85,B 0,C 180,E1 -23786.804,E2 -23786.804} C_VEL
LIN {X 0,Y 244.491,Z 422.765,A -85,B 0,C 180,E1 -23787.988,E2 -23787.988} C_VEL
LIN {X 0,Y 238.948,Z 487.126,A -85,B 0,C 180,E1 -23789.484,E2 -23789.484} C_VEL
LIN {X 0,Y 238.155,Z 492.98,A -85,B 0,C 180,E1 -23789.495,E2 -23789.495} C_VEL
LIN {X 0,Y 233.382,Z 512.029,A -85,B 0,C 180,E1 -23788.812,E2 -23788.812} C_VEL
LIN {X 0,Y 232.124,Z 517.805,A -85,B 0,C 180,E1 -23788.86,E2 -23788.86} C_VEL
LIN {X 0,Y 228.44,Z 535.391,A -85,B 0,C 180,E1 -23789.592,E2 -23789.592} C_VEL
LIN {X 0,Y 223.889,Z 551.565,A -85,B 0,C 180,E1 -23790.54,E2 -23790.54} C_VEL
LIN {X 0,Y 218.873,Z 566.144,A -85,B 0,C 180,E1 -23791.69,E2 -23791.69} C_VEL
LIN {X 0,Y 213.006,Z 580.62,A -85,B 0,C 180,E1 -23793.152,E2 -23793.152} C_VEL
LIN {X 0,Y 206.654,Z 594.138,A -85,B 0,C 180,E1 -23794.871,E2 -23794.871} C_VEL
LIN {X 0,Y 199.367,Z 607.736,A -85,B 0,C 180,E1 -23797.102,E2 -23797.102} C_VEL
LIN {X 0,Y 191.715,Z 620.232,A -85,B 0,C 180,E1 -23799.662,E2 -23799.662} C_VEL
LIN {X 0,Y 184.124,Z 631.719,A -85,B 0,C 180,E1 -23802.713,E2 -23802.713} C_VEL
LIN {X 0,Y 177.157,Z 641.585,A -85,B 0,C 180,E1 -23806.034,E2 -23806.034} C_VEL
LIN {X 0,Y 169.825,Z 651.081,A -85,B 0,C 180,E1 -23810.101,E2 -23810.101} C_VEL
LIN {X 0,Y 162.702,Z 660.031,A -85,B 0,C 180,E1 -23815.156,E2 -23815.156} C_VEL
LIN {X 0,Y 156.974,Z 667.122,A -85,B 0,C 180,E1 -23820.496,E2 -23820.496} C_VEL
LIN {X 0,Y 153.03,Z 672.264,A -85,B 0,C 180,E1 -23825.586,E2 -23825.586} C_VEL
LIN {X 0,Y 150.203,Z 676.274,A -85,B 0,C 180,E1 -23830.881,E2 -23830.881} C_VEL
LIN {X 0,Y 148.351,Z 679.245,A -85,B 0,C 180,E1 -23836.298,E2 -23836.298} C_VEL
LIN {X 0,Y 147.608,Z 681.216,A -85,B 0,C 180,E1 -23841.788,E2 -23841.788} C_VEL
LIN {X 0,Y 147.565,Z 682.196,A -85,B 0,C 180,E1 -23847.27,E2 -23847.27} C_VEL
LIN {X 0,Y 147.715,Z 682.356,A -85,B 0,C 180,E1 -23850,E2 -23850} C_VEL
LIN {X 0,Y 147.538,Z 681.801,A -85,B 0,C 180,E1 -23855.467,E2 -23855.467} C_VEL
LIN {X 0,Y 147.888,Z 680.357,A -85,B 0,C 180,E1 -23860.958,E2 -23860.958} C_VEL
LIN {X 0,Y 149.14,Z 677.83,A -85,B 0,C 180,E1 -23866.424,E2 -23866.424} C_VEL
LIN {X 0,Y 151.652,Z 674.152,A -85,B 0,C 180,E1 -23872.051,E2 -23872.051} C_VEL
LIN {X 0,Y 155.915,Z 668.478,A -85,B 0,C 180,E1 -23878.248,E2 -23878.248} C_VEL
LIN {X 0,Y 162.082,Z 660.75,A -85,B 0,C 180,E1 -23884.311,E2 -23884.311} C_VEL
LIN {X 0,Y 169.013,Z 652.051,A -85,B 0,C 180,E1 -23889.356,E2 -23889.356} C_VEL
LIN {X 0,Y 176.128,Z 642.684,A -85,B 0,C 180,E1 -23893.487,E2 -23893.487} C_VEL
LIN {X 0,Y 183.057,Z 633.021,A -85,B 0,C 180,E1 -23896.84,E2 -23896.84} C_VEL
LIN {X 0,Y 190.584,Z 621.788,A -85,B 0,C 180,E1 -23899.922,E2 -23899.922} C_VEL
LIN {X 0,Y 197.5,Z 610.61,A -85,B 0,C 180,E1 -23902.323,E2 -23902.323} C_VEL
LIN {X 0,Y 204.662,Z 597.618,A -85,B 0,C 180,E1 -23904.558,E2 -23904.558} C_VEL
LIN {X 0,Y 211.719,Z 583.097,A -85,B 0,C 180,E1 -23906.513,E2 -23906.513} C_VEL
LIN {X 0,Y 217.575,Z 569.202,A -85,B 0,C 180,E1 -23907.985,E2 -23907.985} C_VEL
LIN {X 0,Y 223.21,Z 553.187,A -85,B 0,C 180,E1 -23909.312,E2 -23909.312} C_VEL
LIN {X 0,Y 227.794,Z 536.943,A -85,B 0,C 180,E1 -23910.311,E2 -23910.311} C_VEL
LIN {X 0,Y 231.351,Z 520.783,A -85,B 0,C 180,E1 -23911,E2 -23911} C_VEL
LIN {X 0,Y 233.728,Z 504.555,A -85,B 0,C 180,E1 -23911.535,E2 -23911.535} C_VEL
LIN {X 0,Y 240.72,Z 425.694,A -85,B 0,C 180,E1 -23913.416,E2 -23913.416} C_VEL
LIN {X 0,Y 236.668,Z 415.849,A -85,B 0,C 180,E1 -23916.134,E2 -23916.134} C_VEL
LIN {X 0,Y 234.625,Z 411.408,A -85,B 0,C 180,E1 -23917.62,E2 -23917.62} C_VEL
LIN {X 0,Y 230.444,Z 403.994,A -85,B 0,C 180,E1 -23920.937,E2 -23920.937} C_VEL
LIN {X 0,Y 227.774,Z 399.641,A -85,B 0,C 180,E1 -23923.417,E2 -23923.417} C_VEL
LIN {X 0,Y 225.781,Z 396.349,A -85,B 0,C 180,E1 -23925.581,E2 -23925.581} C_VEL
LIN {X 0,Y 223.773,Z 392.969,A -85,B 0,C 180,E1 -23928.199,E2 -23928.199} C_VEL
LIN {X 0,Y 221.685,Z 389.458,A -85,B 0,C 180,E1 -23931.798,E2 -23931.798} C_VEL
LIN {X 0,Y 221.292,Z 388.678,A -85,B 0,C 180,E1 -23932.702,E2 -23932.702} C_VEL
LIN {X 0,Y 219.708,Z 386.067,A -85,B 0,C 180,E1 -23940,E2 -23940} C_VEL
LIN {X 0,Y 221.501,Z 388.928,A -85,B 0,C 180,E1 -23948.209,E2 -23948.209} C_VEL
LIN {X 0,Y 223.522,Z 392.685,A -85,B 0,C 180,E1 -23951.908,E2 -23951.908} C_VEL
LIN {X 0,Y 224.388,Z 394.039,A -85,B 0,C 180,E1 -23953.125,E2 -23953.125} C_VEL
LIN {X 0,Y 227.008,Z 398.326,A -85,B 0,C 180,E1 -23956.24,E2 -23956.24} C_VEL
LIN {X 0,Y 229.575,Z 402.547,A -85,B 0,C 180,E1 -23958.75,E2 -23958.75} C_VEL
LIN {X 0,Y 233.138,Z 408.811,A -85,B 0,C 180,E1 -23961.729,E2 -23961.729} C_VEL
LIN {X 0,Y 237.392,Z 416.552,A -85,B 0,C 180,E1 -23964.76,E2 -23964.76} C_VEL
LIN {X 0,Y 240.797,Z 423.45,A -85,B 0,C 180,E1 -23966.93,E2 -23966.93} C_VEL
LIN {X 0,Y 233.952,Z 500.809,A -85,B 0,C 180,E1 -23968.819,E2 -23968.819} C_VEL
LIN {X 0,Y 231.271,Z 517.779,A -85,B 0,C 180,E1 -23969.446,E2 -23969.446} C_VEL
LIN {X 0,Y 227.773,Z 533.311,A -85,B 0,C 180,E1 -23970.238,E2 -23970.238} C_VEL
LIN {X 0,Y 223.863,Z 547.281,A -85,B 0,C 180,E1 -23971.187,E2 -23971.187} C_VEL
LIN {X 0,Y 218.658,Z 562.224,A -85,B 0,C 180,E1 -23972.466,E2 -23972.466} C_VEL
LIN {X 0,Y 212.971,Z 576.06,A -85,B 0,C 180,E1 -23973.992,E2 -23973.992} C_VEL
LIN {X 0,Y 206.264,Z 590.255,A -85,B 0,C 180,E1 -23975.98,E2 -23975.98} C_VEL
LIN {X 0,Y 199.07,Z 603.32,A -85,B 0,C 180,E1 -23978.232,E2 -23978.232} C_VEL
LIN {X 0,Y 192.383,Z 614.444,A -85,B 0,C 180,E1 -23980.71,E2 -23980.71} C_VEL
LIN {X 0,Y 184.971,Z 625.544,A -85,B 0,C 180,E1 -23983.788,E2 -23983.788} C_VEL
LIN {X 0,Y 177.112,Z 636.28,A -85,B 0,C 180,E1 -23987.579,E2 -23987.579} C_VEL
LIN {X 0,Y 169.915,Z 645.485,A -85,B 0,C 180,E1 -23991.802,E2 -23991.802} C_VEL
LIN {X 0,Y 163.908,Z 652.813,A -85,B 0,C 180,E1 -23996.123,E2 -23996.123} C_VEL
LIN {X 0,Y 157.596,Z 660.36,A -85,B 0,C 180,E1 -24002.079,E2 -24002.079} C_VEL
LIN {X 0,Y 152.886,Z 666.079,A -85,B 0,C 180,E1 -24008.423,E2 -24008.423} C_VEL
LIN {X 0,Y 150.18,Z 669.422,A -85,B 0,C 180,E1 -24013.693,E2 -24013.693} C_VEL
LIN {X 0,Y 148.615,Z 671.841,A -85,B 0,C 180,E1 -24019.096,E2 -24019.096} C_VEL
LIN {X 0,Y 147.856,Z 673.207,A -85,B 0,C 180,E1 -24024.545,E2 -24024.545} C_VEL
LIN {X 0,Y 147.766,Z 673.728,A -85,B 0,C 180,E1 -24030,E2 -24030} C_VEL
LIN {X 0,Y 147.856,Z 673.238,A -85,B 0,C 180,E1 -24035.455,E2 -24035.455} C_VEL
LIN {X 0,Y 148.609,Z 671.902,A -85,B 0,C 180,E1 -24040.904,E2 -24040.904} C_VEL
LIN {X 0,Y 150.154,Z 669.513,A -85,B 0,C 180,E1 -24046.31,E2 -24046.31} C_VEL
LIN {X 0,Y 152.808,Z 666.209,A -85,B 0,C 180,E1 -24051.588,E2 -24051.588} C_VEL
LIN {X 0,Y 157.569,Z 660.524,A -85,B 0,C 180,E1 -24057.925,E2 -24057.925} C_VEL
LIN {X 0,Y 163.864,Z 653.034,A -85,B 0,C 180,E1 -24063.887,E2 -24063.887} C_VEL
LIN {X 0,Y 170.817,Z 644.541,A -85,B 0,C 180,E1 -24068.861,E2 -24068.861} C_VEL
LIN {X 0,Y 177.977,Z 635.361,A -85,B 0,C 180,E1 -24072.935,E2 -24072.935} C_VEL
LIN {X 0,Y 185.669,Z 624.8,A -85,B 0,C 180,E1 -24076.576,E2 -24076.576} C_VEL
LIN {X 0,Y 192.275,Z 614.88,A -85,B 0,C 180,E1 -24079.327,E2 -24079.327} C_VEL
LIN {X 0,Y 200.206,Z 601.823,A -85,B 0,C 180,E1 -24082.169,E2 -24082.169} C_VEL
LIN {X 0,Y 207.963,Z 587.342,A -85,B 0,C 180,E1 -24084.603,E2 -24084.603} C_VEL
LIN {X 0,Y 214.094,Z 573.91,A -85,B 0,C 180,E1 -24086.405,E2 -24086.405} C_VEL
LIN {X 0,Y 219.851,Z 559.559,A -85,B 0,C 180,E1 -24087.9,E2 -24087.9} C_VEL
LIN {X 0,Y 225.058,Z 543.979,A -85,B 0,C 180,E1 -24089.176,E2 -24089.176} C_VEL
LIN {X 0,Y 229.225,Z 528.224,A -85,B 0,C 180,E1 -24090.191,E2 -24090.191} C_VEL
LIN {X 0,Y 232.633,Z 511.416,A -85,B 0,C 180,E1 -24090.937,E2 -24090.937} C_VEL
LIN {X 0,Y 234.74,Z 495.182,A -85,B 0,C 180,E1 -24091.461,E2 -24091.461} C_VEL
LIN {X 0,Y 241.014,Z 423.661,A -85,B 0,C 180,E1 -24093.172,E2 -24093.172} C_VEL
LIN {X 0,Y 236.374,Z 414.401,A -85,B 0,C 180,E1 -24096.188,E2 -24096.188} C_VEL
LIN {X 0,Y 232.157,Z 406.855,A -85,B 0,C 180,E1 -24099.337,E2 -24099.337} C_VEL
LIN {X 0,Y 228.769,Z 400.945,A -85,B 0,C 180,E1 -24102.34,E2 -24102.34} C_VEL
LIN {X 0,Y 226.01,Z 396.571,A -85,B 0,C 180,E1 -24105.25,E2 -24105.25} C_VEL
LIN {X 0,Y 223.935,Z 393.044,A -85,B 0,C 180,E1 -24107.986,E2 -24107.986} C_VEL
LIN {X 0,Y 221.943,Z 389.832,A -85,B 0,C 180,E1 -24111.435,E2 -24111.435} C_VEL
LIN {X 0,Y 221.618,Z 388.874,A -85,B 0,C 180,E1 -24112.254,E2 -24112.254} C_VEL
LIN {X 0,Y 219.979,Z 386.528,A -85,B 0,C 180,E1 -24120,E2 -24120} C_VEL
LIN {X 0,Y 221.713,Z 389.148,A -85,B 0,C 180,E1 -24127.628,E2 -24127.628} C_VEL
LIN {X 0,Y 223.407,Z 392.407,A -85,B 0,C 180,E1 -24130.88,E2 -24130.88} C_VEL
LIN {X 0,Y 224.479,Z 393.981,A -85,B 0,C 180,E1 -24132.429,E2 -24132.429} C_VEL
LIN {X 0,Y 227.088,Z 398.315,A -85,B 0,C 180,E1 -24135.596,E2 -24135.596} C_VEL
LIN {X 0,Y 230.151,Z 403.346,A -85,B 0,C 180,E1 -24138.585,E2 -24138.585} C_VEL
LIN {X 0,Y 234.162,Z 410.412,A -85,B 0,C 180,E1 -24141.86,E2 -24141.86} C_VEL
LIN {X 0,Y 236.533,Z 415.14,A -85,B 0,C 180,E1 -24143.589,E2 -24143.589} C_VEL
LIN {X 0,Y 240.731,Z 425.333,A -85,B 0,C 180,E1 -24146.437,E2 -24146.437} C_VEL
LIN {X 0,Y 240.918,Z 425.824,A -85,B 0,C 180,E1 -24146.557,E2 -24146.557} C_VEL
LIN {X 0,Y 233.666,Z 507.089,A -85,B 0,C 180,E1 -24148.503,E2 -24148.503} C_VEL
LIN {X 0,Y 232.124,Z 517.805,A -85,B 0,C 180,E1 -24148.86,E2 -24148.86} C_VEL
LIN {X 0,Y 230.704,Z 523.542,A -85,B 0,C 180,E1 -24148.916,E2 -24148.916} C_VEL
LIN {X 0,Y 223.867,Z 541.055,A -85,B 0,C 180,E1 -24148.518,E2 -24148.518} C_VEL
LIN {X 0,Y 222.164,Z 545.678,A -85,B 0,C 180,E1 -24148.608,E2 -24148.608} C_VEL
LIN {X 0,Y 221.568,Z 547.476,A -85,B 0,C 180,E1 -24148.704,E2 -24148.704} C_VEL
LIN {X 0,Y 216.589,Z 562.403,A -85,B 0,C 180,E1 -24149.774,E2 -24149.774} C_VEL
LIN {X 0,Y 210.53,Z 577.474,A -85,B 0,C 180,E1 -24151.195,E2 -24151.195} C_VEL
LIN {X 0,Y 203.935,Z 591.343,A -85,B 0,C 180,E1 -24152.86,E2 -24152.86} C_VEL
LIN {X 0,Y 196.946,Z 604.308,A -85,B 0,C 180,E1 -24154.841,E2 -24154.841} C_VEL
LIN {X 0,Y 189.626,Z 616.445,A -85,B 0,C 180,E1 -24157.171,E2 -24157.171} C_VEL
LIN {X 0,Y 181.545,Z 628.452,A -85,B 0,C 180,E1 -24160.133,E2 -24160.133} C_VEL
LIN {X 0,Y 173.225,Z 639.712,A -85,B 0,C 180,E1 -24163.737,E2 -24163.737} C_VEL
LIN {X 0,Y 166.188,Z 648.619,A -85,B 0,C 180,E1 -24167.42,E2 -24167.42} C_VEL
LIN {X 0,Y 159.242,Z 656.996,A -85,B 0,C 180,E1 -24171.839,E2 -24171.839} C_VEL
LIN {X 0,Y 153.292,Z 663.93,A -85,B 0,C 180,E1 -24176.622,E2 -24176.622} C_VEL
LIN {X 0,Y 148.474,Z 669.616,A -85,B 0,C 180,E1 -24181.749,E2 -24181.749} C_VEL
LIN {X 0,Y 144.815,Z 674.276,A -85,B 0,C 180,E1 -24187.231,E2 -24187.231} C_VEL
LIN {X 0,Y 142.274,Z 677.666,A -85,B 0,C 180,E1 -24192.76,E2 -24192.76} C_VEL
LIN {X 0,Y 140.846,Z 680.178,A -85,B 0,C 180,E1 -24198.487,E2 -24198.487} C_VEL
LIN {X 0,Y 140.438,Z 681.608,A -85,B 0,C 180,E1 -24204.256,E2 -24204.256} C_VEL
LIN {X 0,Y 140.627,Z 682.149,A -85,B 0,C 180,E1 -24210,E2 -24210} C_VEL
LIN {X 0,Y 140.438,Z 681.592,A -85,B 0,C 180,E1 -24215.744,E2 -24215.744} C_VEL
LIN {X 0,Y 140.846,Z 680.147,A -85,B 0,C 180,E1 -24221.513,E2 -24221.513} C_VEL
LIN {X 0,Y 142.271,Z 677.62,A -85,B 0,C 180,E1 -24227.241,E2 -24227.241} C_VEL
LIN {X 0,Y 144.847,Z 674.161,A -85,B 0,C 180,E1 -24232.84,E2 -24232.84} C_VEL
LIN {X 0,Y 149.591,Z 668.266,A -85,B 0,C 180,E1 -24239.558,E2 -24239.558} C_VEL
LIN {X 0,Y 156.189,Z 660.538,A -85,B 0,C 180,E1 -24245.8,E2 -24245.8} C_VEL
LIN {X 0,Y 163.497,Z 651.838,A -85,B 0,C 180,E1 -24250.959,E2 -24250.959} C_VEL
LIN {X 0,Y 170.846,Z 642.624,A -85,B 0,C 180,E1 -24255.089,E2 -24255.089} C_VEL
LIN {X 0,Y 178.221,Z 632.809,A -85,B 0,C 180,E1 -24258.525,E2 -24258.525} C_VEL
LIN {X 0,Y 186.027,Z 621.575,A -85,B 0,C 180,E1 -24261.621,E2 -24261.621} C_VEL
LIN {X 0,Y 194.193,Z 608.798,A -85,B 0,C 180,E1 -24264.314,E2 -24264.314} C_VEL
LIN {X 0,Y 201.313,Z 596.111,A -85,B 0,C 180,E1 -24266.414,E2 -24266.414} C_VEL
LIN {X 0,Y 207.86,Z 582.884,A -85,B 0,C 180,E1 -24268.158,E2 -24268.158} C_VEL
LIN {X 0,Y 213.888,Z 568.989,A -85,B 0,C 180,E1 -24269.601,E2 -24269.601} C_VEL
LIN {X 0,Y 219.672,Z 552.974,A -85,B 0,C 180,E1 -24270.904,E2 -24270.904} C_VEL
LIN {X 0,Y 224.008,Z 538.054,A -85,B 0,C 180,E1 -24271.813,E2 -24271.813} C_VEL
LIN {X 0,Y 227.724,Z 521.897,A -85,B 0,C 180,E1 -24272.517,E2 -24272.517} C_VEL
LIN {X 0,Y 230.341,Z 505.172,A -85,B 0,C 180,E1 -24273.063,E2 -24273.063} C_VEL
LIN {X 0,Y 237.271,Z 428.873,A -85,B 0,C 180,E1 -24274.893,E2 -24274.893} C_VEL
LIN {X 0,Y 233.41,Z 419.222,A -85,B 0,C 180,E1 -24277.723,E2 -24277.723} C_VEL
LIN {X 0,Y 230.094,Z 412.917,A -85,B 0,C 180,E1 -24280.368,E2 -24280.368} C_VEL
LIN {X 0,Y 226.889,Z 407.158,A -85,B 0,C 180,E1 -24283.35,E2 -24283.35} C_VEL
LIN {X 0,Y 224.412,Z 402.995,A -85,B 0,C 180,E1 -24286.104,E2 -24286.104} C_VEL
LIN {X 0,Y 222.584,Z 399.786,A -85,B 0,C 180,E1 -24288.608,E2 -24288.608} C_VEL
LIN {X 0,Y 220.602,Z 396.295,A -85,B 0,C 180,E1 -24292.219,E2 -24292.219} C_VEL
LIN {X 0,Y 220.226,Z 395.59,A -85,B 0,C 180,E1 -24293.127,E2 -24293.127} C_VEL
LIN {X 0,Y 218.839,Z 393.147,A -85,B 0,C 180,E1 -24300,E2 -24300} C_VEL
LIN {X 0,Y 220.472,Z 395.911,A -85,B 0,C 180,E1 -24307.902,E2 -24307.902} C_VEL
LIN {X 0,Y 222.582,Z 399.775,A -85,B 0,C 180,E1 -24311.844,E2 -24311.844} C_VEL
LIN {X 0,Y 225.532,Z 404.902,A -85,B 0,C 180,E1 -24315.667,E2 -24315.667} C_VEL
LIN {X 0,Y 228.159,Z 409.432,A -85,B 0,C 180,E1 -24318.353,E2 -24318.353} C_VEL
LIN {X 0,Y 231.624,Z 415.783,A -85,B 0,C 180,E1 -24321.353,E2 -24321.353} C_VEL
LIN {X 0,Y 235.362,Z 422.958,A -85,B 0,C 180,E1 -24324.13,E2 -24324.13} C_VEL
LIN {X 0,Y 237.376,Z 427.141,A -85,B 0,C 180,E1 -24325.497,E2 -24325.497} C_VEL
LIN {X 0,Y 230.699,Z 500.422,A -85,B 0,C 180,E1 -24327.266,E2 -24327.266} C_VEL
LIN {X 0,Y 228.044,Z 517.083,A -85,B 0,C 180,E1 -24327.859,E2 -24327.859} C_VEL
LIN {X 0,Y 224.286,Z 533.526,A -85,B 0,C 180,E1 -24328.673,E2 -24328.673} C_VEL
LIN {X 0,Y 219.608,Z 549.474,A -85,B 0,C 180,E1 -24329.766,E2 -24329.766} C_VEL
LIN {X 0,Y 214.259,Z 564.142,A -85,B 0,C 180,E1 -24331.026,E2 -24331.026} C_VEL
LIN {X 0,Y 207.768,Z 579.168,A -85,B 0,C 180,E1 -24332.726,E2 -24332.726} C_VEL
LIN {X 0,Y 200.928,Z 592.802,A -85,B 0,C 180,E1 -24334.717,E2 -24334.717} C_VEL
LIN {X 0,Y 193.568,Z 605.47,A -85,B 0,C 180,E1 -24336.988,E2 -24336.988} C_VEL
LIN {X 0,Y 186.679,Z 616.386,A -85,B 0,C 180,E1 -24339.487,E2 -24339.487} C_VEL
LIN {X 0,Y 179.023,Z 627.23,A -85,B 0,C 180,E1 -24342.602,E2 -24342.602} C_VEL
LIN {X 0,Y 171.913,Z 636.49,A -85,B 0,C 180,E1 -24345.975,E2 -24345.975} C_VEL
LIN {X 0,Y 164.489,Z 645.5,A -85,B 0,C 180,E1 -24350.142,E2 -24350.142} C_VEL
LIN {X 0,Y 158.016,Z 653.024,A -85,B 0,C 180,E1 -24354.677,E2 -24354.677} C_VEL
LIN {X 0,Y 151.292,Z 660.57,A -85,B 0,C 180,E1 -24360.807,E2 -24360.807} C_VEL
LIN {X 0,Y 147.108,Z 665.241,A -85,B 0,C 180,E1 -24366.041,E2 -24366.041} C_VEL
LIN {X 0,Y 144.668,Z 668.077,A -85,B 0,C 180,E1 -24370.119,E2 -24370.119} C_VEL
LIN {X 0,Y 142.365,Z 670.955,A -85,B 0,C 180,E1 -24375.71,E2 -24375.71} C_VEL
LIN {X 0,Y 141.094,Z 672.839,A -85,B 0,C 180,E1 -24381.406,E2 -24381.406} C_VEL
LIN {X 0,Y 140.653,Z 673.825,A -85,B 0,C 180,E1 -24387.923,E2 -24387.923} C_VEL
LIN {X 0,Y 140.653,Z 673.835,A -85,B 0,C 180,E1 -24392.077,E2 -24392.077} C_VEL
LIN {X 0,Y 141.092,Z 672.89,A -85,B 0,C 180,E1 -24398.594,E2 -24398.594} C_VEL
LIN {X 0,Y 142.349,Z 671.026,A -85,B 0,C 180,E1 -24404.291,E2 -24404.291} C_VEL
LIN {X 0,Y 144.627,Z 668.187,A -85,B 0,C 180,E1 -24409.886,E2 -24409.886} C_VEL
LIN {X 0,Y 148.512,Z 663.793,A -85,B 0,C 180,E1 -24415.955,E2 -24415.955} C_VEL
LIN {X 0,Y 153.746,Z 657.934,A -85,B 0,C 180,E1 -24421.714,E2 -24421.714} C_VEL
LIN {X 0,Y 159.531,Z 651.454,A -85,B 0,C 180,E1 -24426.493,E2 -24426.493} C_VEL
LIN {X 0,Y 166.169,Z 643.677,A -85,B 0,C 180,E1 -24430.962,E2 -24430.962} C_VEL
LIN {X 0,Y 173.788,Z 634.347,A -85,B 0,C 180,E1 -24435.048,E2 -24435.048} C_VEL
LIN {X 0,Y 181.242,Z 624.411,A -85,B 0,C 180,E1 -24438.413,E2 -24438.413} C_VEL
LIN {X 0,Y 188.849,Z 613.315,A -85,B 0,C 180,E1 -24441.398,E2 -24441.398} C_VEL
LIN {X 0,Y 196.542,Z 600.964,A -85,B 0,C 180,E1 -24444,E2 -24444} C_VEL
LIN {X 0,Y 203.3,Z 588.692,A -85,B 0,C 180,E1 -24446.064,E2 -24446.064} C_VEL
LIN {X 0,Y 209.592,Z 575.534,A -85,B 0,C 180,E1 -24447.851,E2 -24447.851} C_VEL
LIN {X 0,Y 216.163,Z 559.76,A -85,B 0,C 180,E1 -24449.494,E2 -24449.494} C_VEL
LIN {X 0,Y 221.494,Z 544.179,A -85,B 0,C 180,E1 -24450.758,E2 -24450.758} C_VEL
LIN {X 0,Y 225.741,Z 528.64,A -85,B 0,C 180,E1 -24451.738,E2 -24451.738} C_VEL
LIN {X 0,Y 229.211,Z 511.957,A -85,B 0,C 180,E1 -24452.47,E2 -24452.47} C_VEL
LIN {X 0,Y 231.417,Z 495.566,A -85,B 0,C 180,E1 -24452.996,E2 -24452.996} C_VEL
LIN {X 0,Y 237.538,Z 427.969,A -85,B 0,C 180,E1 -24454.594,E2 -24454.594} C_VEL
LIN {X 0,Y 237.453,Z 427.048,A -85,B 0,C 180,E1 -24454.702,E2 -24454.702} C_VEL
LIN {X 0,Y 233.694,Z 419.455,A -85,B 0,C 180,E1 -24457.336,E2 -24457.336} C_VEL
LIN {X 0,Y 230.103,Z 412.748,A -85,B 0,C 180,E1 -24460.208,E2 -24460.208} C_VEL
LIN {X 0,Y 227.006,Z 407.173,A -85,B 0,C 180,E1 -24463.127,E2 -24463.127} C_VEL
LIN {X 0,Y 224.751,Z 403.402,A -85,B 0,C 180,E1 -24465.64,E2 -24465.64} C_VEL
LIN {X 0,Y 222.68,Z 399.78,A -85,B 0,C 180,E1 -24468.501,E2 -24468.501} C_VEL
LIN {X 0,Y 220.764,Z 396.37,A -85,B 0,C 180,E1 -24472.109,E2 -24472.109} C_VEL
LIN {X 0,Y 220.357,Z 395.643,A -85,B 0,C 180,E1 -24473.131,E2 -24473.131} C_VEL
LIN {X 0,Y 219.113,Z 393.578,A -85,B 0,C 180,E1 -24480,E2 -24480} C_VEL
LIN {X 0,Y 220.651,Z 395.96,A -85,B 0,C 180,E1 -24487.204,E2 -24487.204} C_VEL
LIN {X 0,Y 222.251,Z 399.244,A -85,B 0,C 180,E1 -24490.476,E2 -24490.476} C_VEL
LIN {X 0,Y 223.277,Z 400.856,A -85,B 0,C 180,E1 -24492.036,E2 -24492.036} C_VEL
LIN {X 0,Y 225.652,Z 404.958,A -85,B 0,C 180,E1 -24495.058,E2 -24495.058} C_VEL
LIN {X 0,Y 228.154,Z 409.23,A -85,B 0,C 180,E1 -24497.651,E2 -24497.651} C_VEL
LIN {X 0,Y 231.194,Z 414.746,A -85,B 0,C 180,E1 -24500.345,E2 -24500.345} C_VEL
LIN {X 0,Y 233.765,Z 419.735,A -85,B 0,C 180,E1 -24502.362,E2 -24502.362} C_VEL
LIN {X 0,Y 237.357,Z 428.725,A -85,B 0,C 180,E1 -24505,E2 -24505} C_VEL
LIN {X 0,Y 237.52,Z 429.157,A -85,B 0,C 180,E1 -24505.113,E2 -24505.113} C_VEL
LIN {X 0,Y 230.278,Z 507.622,A -85,B 0,C 180,E1 -24506.97,E2 -24506.97} C_VEL
LIN {X 0,Y 227.625,Z 523.479,A -85,B 0,C 180,E1 -24507.509,E2 -24507.509} C_VEL
LIN {X 0,Y 223.907,Z 539.356,A -85,B 0,C 180,E1 -24508.245,E2 -24508.245} C_VEL
LIN {X 0,Y 221.568,Z 547.476,A -85,B 0,C 180,E1 -24508.704,E2 -24508.704} C_VEL
LIN {X 0,Y 219.529,Z 553.065,A -85,B 0,C 180,E1 -24508.921,E2 -24508.921} C_VEL
LIN {X 0,Y 211.117,Z 568.846,A -85,B 0,C 180,E1 -24508.962,E2 -24508.962} C_VEL
LIN {X 0,Y 208.435,Z 573.917,A -85,B 0,C 180,E1 -24509.198,E2 -24509.198} C_VEL
LIN {X 0,Y 207.658,Z 575.601,A -85,B 0,C 180,E1 -24509.343,E2 -24509.343} C_VEL
LIN {X 0,Y 200.823,Z 589.843,A -85,B 0,C 180,E1 -24510.975,E2 -24510.975} C_VEL
LIN {X 0,Y 193.597,Z 603.029,A -85,B 0,C 180,E1 -24512.915,E2 -24512.915} C_VEL
LIN {X 0,Y 185.398,Z 616.24,A -85,B 0,C 180,E1 -24515.412,E2 -24515.412} C_VEL
LIN {X 0,Y 176.998,Z 628.245,A -85,B 0,C 180,E1 -24518.353,E2 -24518.353} C_VEL
LIN {X 0,Y 168.69,Z 639.048,A -85,B 0,C 180,E1 -24521.804,E2 -24521.804} C_VEL
LIN {X 0,Y 160.979,Z 648.411,A -85,B 0,C 180,E1 -24525.692,E2 -24525.692} C_VEL
LIN {X 0,Y 153.636,Z 656.787,A -85,B 0,C 180,E1 -24530.177,E2 -24530.177} C_VEL
LIN {X 0,Y 147.317,Z 663.72,A -85,B 0,C 180,E1 -24535.077,E2 -24535.077} C_VEL
LIN {X 0,Y 142.172,Z 669.407,A -85,B 0,C 180,E1 -24540.375,E2 -24540.375} C_VEL
LIN {X 0,Y 137.934,Z 674.353,A -85,B 0,C 180,E1 -24546.51,E2 -24546.51} C_VEL
LIN {X 0,Y 135.443,Z 677.457,A -85,B 0,C 180,E1 -24551.861,E2 -24551.861} C_VEL
LIN {X 0,Y 133.827,Z 679.969,A -85,B 0,C 180,E1 -24557.874,E2 -24557.874} C_VEL
LIN {X 0,Y 133.345,Z 681.4,A -85,B 0,C 180,E1 -24563.949,E2 -24563.949} C_VEL
LIN {X 0,Y 133.531,Z 681.942,A -85,B 0,C 180,E1 -24570,E2 -24570} C_VEL
LIN {X 0,Y 133.345,Z 681.384,A -85,B 0,C 180,E1 -24576.051,E2 -24576.051} C_VEL
LIN {X 0,Y 133.826,Z 679.938,A -85,B 0,C 180,E1 -24582.126,E2 -24582.126} C_VEL
LIN {X 0,Y 135.439,Z 677.41,A -85,B 0,C 180,E1 -24588.14,E2 -24588.14} C_VEL
LIN {X 0,Y 138.217,Z 673.949,A -85,B 0,C 180,E1 -24594.003,E2 -24594.003} C_VEL
LIN {X 0,Y 143.35,Z 668.054,A -85,B 0,C 180,E1 -24600.983,E2 -24600.983} C_VEL
LIN {X 0,Y 150.372,Z 660.325,A -85,B 0,C 180,E1 -24607.415,E2 -24607.415} C_VEL
LIN {X 0,Y 158.122,Z 651.626,A -85,B 0,C 180,E1 -24612.673,E2 -24612.673} C_VEL
LIN {X 0,Y 165.766,Z 642.471,A -85,B 0,C 180,E1 -24616.836,E2 -24616.836} C_VEL
LIN {X 0,Y 173.541,Z 632.596,A -85,B 0,C 180,E1 -24620.304,E2 -24620.304} C_VEL
LIN {X 0,Y 181.661,Z 621.363,A -85,B 0,C 180,E1 -24623.394,E2 -24623.394} C_VEL
LIN {X 0,Y 189.83,Z 609.016,A -85,B 0,C 180,E1 -24625.992,E2 -24625.992} C_VEL
LIN {X 0,Y 197.515,Z 595.781,A -85,B 0,C 180,E1 -24628.159,E2 -24628.159} C_VEL
LIN {X 0,Y 204.182,Z 582.671,A -85,B 0,C 180,E1 -24629.86,E2 -24629.86} C_VEL
LIN {X 0,Y 210.382,Z 568.776,A -85,B 0,C 180,E1 -24631.27,E2 -24631.27} C_VEL
LIN {X 0,Y 216.304,Z 552.76,A -85,B 0,C 180,E1 -24632.55,E2 -24632.55} C_VEL
LIN {X 0,Y 221.281,Z 535.883,A -85,B 0,C 180,E1 -24633.541,E2 -24633.541} C_VEL
LIN {X 0,Y 224.904,Z 519.933,A -85,B 0,C 180,E1 -24634.176,E2 -24634.176} C_VEL
LIN {X 0,Y 227.344,Z 503.631,A -85,B 0,C 180,E1 -24634.702,E2 -24634.702} C_VEL
LIN {X 0,Y 234.011,Z 432.322,A -85,B 0,C 180,E1 -24636.377,E2 -24636.377} C_VEL
LIN {X 0,Y 230.88,Z 424.223,A -85,B 0,C 180,E1 -24638.868,E2 -24638.868} C_VEL
LIN {X 0,Y 227.187,Z 417.014,A -85,B 0,C 180,E1 -24642.097,E2 -24642.097} C_VEL
LIN {X 0,Y 224.563,Z 412.372,A -85,B 0,C 180,E1 -24644.805,E2 -24644.805} C_VEL
LIN {X 0,Y 223.065,Z 409.693,A -85,B 0,C 180,E1 -24646.622,E2 -24646.622} C_VEL
LIN {X 0,Y 221.261,Z 406.413,A -85,B 0,C 180,E1 -24649.245,E2 -24649.245} C_VEL
LIN {X 0,Y 219.366,Z 402.65,A -85,B 0,C 180,E1 -24653.1,E2 -24653.1} C_VEL
LIN {X 0,Y 217.97,Z 400.223,A -85,B 0,C 180,E1 -24660,E2 -24660} C_VEL
LIN {X 0,Y 219.453,Z 402.874,A -85,B 0,C 180,E1 -24667.591,E2 -24667.591} C_VEL
LIN {X 0,Y 221.841,Z 407.433,A -85,B 0,C 180,E1 -24672.116,E2 -24672.116} C_VEL
LIN {X 0,Y 224.173,Z 411.663,A -85,B 0,C 180,E1 -24675.2,E2 -24675.2} C_VEL
LIN {X 0,Y 226.583,Z 415.954,A -85,B 0,C 180,E1 -24677.778,E2 -24677.778} C_VEL
LIN {X 0,Y 230.315,Z 423.085,A -85,B 0,C 180,E1 -24681.128,E2 -24681.128} C_VEL
LIN {X 0,Y 233.908,Z 430.498,A -85,B 0,C 180,E1 -24683.885,E2 -24683.885} C_VEL
LIN {X 0,Y 234.071,Z 430.822,A -85,B 0,C 180,E1 -24684,E2 -24684} C_VEL
LIN {X 0,Y 227.461,Z 501.277,A -85,B 0,C 180,E1 -24685.692,E2 -24685.692} C_VEL
LIN {X 0,Y 224.652,Z 518.216,A -85,B 0,C 180,E1 -24686.302,E2 -24686.302} C_VEL
LIN {X 0,Y 220.97,Z 533.742,A -85,B 0,C 180,E1 -24687.059,E2 -24687.059} C_VEL
LIN {X 0,Y 216.177,Z 549.687,A -85,B 0,C 180,E1 -24688.135,E2 -24688.135} C_VEL
LIN {X 0,Y 210.697,Z 564.354,A -85,B 0,C 180,E1 -24689.376,E2 -24689.376} C_VEL
LIN {X 0,Y 203.989,Z 579.418,A -85,B 0,C 180,E1 -24691.048,E2 -24691.048} C_VEL
LIN {X 0,Y 196.966,Z 593.013,A -85,B 0,C 180,E1 -24693.018,E2 -24693.018} C_VEL
LIN {X 0,Y 189.361,Z 605.681,A -85,B 0,C 180,E1 -24695.263,E2 -24695.263} C_VEL
LIN {X 0,Y 182.219,Z 616.597,A -85,B 0,C 180,E1 -24697.753,E2 -24697.753} C_VEL
LIN {X 0,Y 174.276,Z 627.441,A -85,B 0,C 180,E1 -24700.877,E2 -24700.877} C_VEL
LIN {X 0,Y 166.852,Z 636.701,A -85,B 0,C 180,E1 -24704.27,E2 -24704.27} C_VEL
LIN {X 0,Y 159.049,Z 645.711,A -85,B 0,C 180,E1 -24708.486,E2 -24708.486} C_VEL
LIN {X 0,Y 152.241,Z 653.234,A -85,B 0,C 180,E1 -24713.121,E2 -24713.121} C_VEL
LIN {X 0,Y 145.088,Z 660.78,A -85,B 0,C 180,E1 -24719.429,E2 -24719.429} C_VEL
LIN {X 0,Y 140.604,Z 665.451,A -85,B 0,C 180,E1 -24724.858,E2 -24724.858} C_VEL
LIN {X 0,Y 137.953,Z 668.287,A -85,B 0,C 180,E1 -24729.108,E2 -24729.108} C_VEL
LIN {X 0,Y 135.444,Z 671.165,A -85,B 0,C 180,E1 -24734.963,E2 -24734.963} C_VEL
LIN {X 0,Y 134.067,Z 673.047,A -85,B 0,C 180,E1 -24740.952,E2 -24740.952} C_VEL
LIN {X 0,Y 133.573,Z 673.991,A -85,B 0,C 180,E1 -24746.984,E2 -24746.984} C_VEL
LIN {X 0,Y 133.56,Z 674.094,A -85,B 0,C 180,E1 -24751.167,E2 -24751.167} C_VEL
LIN {X 0,Y 133.723,Z 673.652,A -85,B 0,C 180,E1 -24756.034,E2 -24756.034} C_VEL
LIN {X 0,Y 134.652,Z 672.317,A -85,B 0,C 180,E1 -24762.05,E2 -24762.05} C_VEL
LIN {X 0,Y 136.481,Z 669.93,A -85,B 0,C 180,E1 -24767.997,E2 -24767.997} C_VEL
LIN {X 0,Y 139.579,Z 666.626,A -85,B 0,C 180,E1 -24773.754,E2 -24773.754} C_VEL
LIN {X 0,Y 145.044,Z 660.941,A -85,B 0,C 180,E1 -24780.582,E2 -24780.582} C_VEL
LIN {X 0,Y 152.193,Z 653.449,A -85,B 0,C 180,E1 -24786.892,E2 -24786.892} C_VEL
LIN {X 0,Y 159.906,Z 644.956,A -85,B 0,C 180,E1 -24792.086,E2 -24792.086} C_VEL
LIN {X 0,Y 167.776,Z 635.775,A -85,B 0,C 180,E1 -24796.268,E2 -24796.268} C_VEL
LIN {X 0,Y 175.314,Z 626.319,A -85,B 0,C 180,E1 -24799.611,E2 -24799.611} C_VEL
LIN {X 0,Y 182.107,Z 616.986,A -85,B 0,C 180,E1 -24802.292,E2 -24802.292} C_VEL
LIN {X 0,Y 189.292,Z 606.143,A -85,B 0,C 180,E1 -24804.766,E2 -24804.766} C_VEL
LIN {X 0,Y 196.893,Z 593.566,A -85,B 0,C 180,E1 -24807.015,E2 -24807.015} C_VEL
LIN {X 0,Y 203.398,Z 581.016,A -85,B 0,C 180,E1 -24808.882,E2 -24808.882} C_VEL
LIN {X 0,Y 209.935,Z 566.677,A -85,B 0,C 180,E1 -24810.504,E2 -24810.504} C_VEL
LIN {X 0,Y 215.408,Z 552.601,A -85,B 0,C 180,E1 -24811.752,E2 -24811.752} C_VEL
LIN {X 0,Y 220.172,Z 537.546,A -85,B 0,C 180,E1 -24812.845,E2 -24812.845} C_VEL
LIN {X 0,Y 224.129,Z 521.636,A -85,B 0,C 180,E1 -24813.69,E2 -24813.69} C_VEL
LIN {X 0,Y 227.108,Z 505.006,A -85,B 0,C 180,E1 -24814.326,E2 -24814.326} C_VEL
LIN {X 0,Y 229.469,Z 483.605,A -85,B 0,C 180,E1 -24814.87,E2 -24814.87} C_VEL
LIN {X 0,Y 234.304,Z 431.022,A -85,B 0,C 180,E1 -24816.1,E2 -24816.1} C_VEL
LIN {X 0,Y 230.531,Z 423.213,A -85,B 0,C 180,E1 -24818.994,E2 -24818.994} C_VEL
LIN {X 0,Y 226.503,Z 415.545,A -85,B 0,C 180,E1 -24822.653,E2 -24822.653} C_VEL
LIN {X 0,Y 223.433,Z 410.117,A -85,B 0,C 180,E1 -24826.123,E2 -24826.123} C_VEL
LIN {X 0,Y 221.442,Z 406.517,A -85,B 0,C 180,E1 -24829.022,E2 -24829.022} C_VEL
LIN {X 0,Y 219.635,Z 402.951,A -85,B 0,C 180,E1 -24832.739,E2 -24832.739} C_VEL
LIN {X 0,Y 218.245,Z 400.645,A -85,B 0,C 180,E1 -24840,E2 -24840} C_VEL
LIN {X 0,Y 219.632,Z 402.963,A -85,B 0,C 180,E1 -24846.892,E2 -24846.892} C_VEL
LIN {X 0,Y 221.383,Z 406.433,A -85,B 0,C 180,E1 -24850.517,E2 -24850.517} C_VEL
LIN {X 0,Y 223.979,Z 411.036,A -85,B 0,C 180,E1 -24854.19,E2 -24854.19} C_VEL
LIN {X 0,Y 226.973,Z 416.458,A -85,B 0,C 180,E1 -24857.455,E2 -24857.455} C_VEL
LIN {X 0,Y 230.591,Z 423.371,A -85,B 0,C 180,E1 -24860.692,E2 -24860.692} C_VEL
LIN {X 0,Y 232.574,Z 428.15,A -85,B 0,C 180,E1 -24862.319,E2 -24862.319} C_VEL
LIN {X 0,Y 234.23,Z 432.472,A -85,B 0,C 180,E1 -24863.601,E2 -24863.601} C_VEL
LIN {X 0,Y 227.191,Z 507.08,A -85,B 0,C 180,E1 -24865.365,E2 -24865.365} C_VEL
LIN {X 0,Y 224.462,Z 523.151,A -85,B 0,C 180,E1 -24865.897,E2 -24865.897} C_VEL
LIN {X 0,Y 221.006,Z 537.799,A -85,B 0,C 180,E1 -24866.547,E2 -24866.547} C_VEL
LIN {X 0,Y 216.297,Z 553.346,A -85,B 0,C 180,E1 -24867.447,E2 -24867.447} C_VEL
LIN {X 0,Y 210.365,Z 569.28,A -85,B 0,C 180,E1 -24868.721,E2 -24868.721} C_VEL
LIN {X 0,Y 207.658,Z 575.601,A -85,B 0,C 180,E1 -24869.343,E2 -24869.343} C_VEL
LIN {X 0,Y 205.018,Z 580.71,A -85,B 0,C 180,E1 -24869.718,E2 -24869.718} C_VEL
LIN {X 0,Y 194.838,Z 595.246,A -85,B 0,C 180,E1 -24870.25,E2 -24870.25} C_VEL
LIN {X 0,Y 191.587,Z 599.96,A -85,B 0,C 180,E1 -24870.676,E2 -24870.676} C_VEL
LIN {X 0,Y 190.621,Z 601.516,A -85,B 0,C 180,E1 -24870.891,E2 -24870.891} C_VEL
LIN {X 0,Y 182.634,Z 614.109,A -85,B 0,C 180,E1 -24873.18,E2 -24873.18} C_VEL
LIN {X 0,Y 175.036,Z 624.763,A -85,B 0,C 180,E1 -24875.603,E2 -24875.603} C_VEL
LIN {X 0,Y 166.734,Z 635.525,A -85,B 0,C 180,E1 -24878.759,E2 -24878.759} C_VEL
LIN {X 0,Y 159.098,Z 644.687,A -85,B 0,C 180,E1 -24882.277,E2 -24882.277} C_VEL
LIN {X 0,Y 150.933,Z 653.587,A -85,B 0,C 180,E1 -24886.622,E2 -24886.622} C_VEL
LIN {X 0,Y 144.125,Z 660.811,A -85,B 0,C 180,E1 -24891.279,E2 -24891.279} C_VEL
LIN {X 0,Y 137.209,Z 667.929,A -85,B 0,C 180,E1 -24897.465,E2 -24897.465} C_VEL
LIN {X 0,Y 131.666,Z 673.804,A -85,B 0,C 180,E1 -24904.722,E2 -24904.722} C_VEL
LIN {X 0,Y 128.636,Z 677.248,A -85,B 0,C 180,E1 -24910.865,E2 -24910.865} C_VEL
LIN {X 0,Y 126.835,Z 679.761,A -85,B 0,C 180,E1 -24917.195,E2 -24917.195} C_VEL
LIN {X 0,Y 126.244,Z 681.191,A -85,B 0,C 180,E1 -24923.608,E2 -24923.608} C_VEL
LIN {X 0,Y 126.426,Z 681.734,A -85,B 0,C 180,E1 -24930,E2 -24930} C_VEL
LIN {X 0,Y 126.244,Z 681.175,A -85,B 0,C 180,E1 -24936.393,E2 -24936.393} C_VEL
LIN {X 0,Y 126.834,Z 679.728,A -85,B 0,C 180,E1 -24942.806,E2 -24942.806} C_VEL
LIN {X 0,Y 128.631,Z 677.2,A -85,B 0,C 180,E1 -24949.137,E2 -24949.137} C_VEL
LIN {X 0,Y 131.666,Z 673.738,A -85,B 0,C 180,E1 -24955.279,E2 -24955.279} C_VEL
LIN {X 0,Y 137.223,Z 667.842,A -85,B 0,C 180,E1 -24962.532,E2 -24962.532} C_VEL
LIN {X 0,Y 144.693,Z 660.112,A -85,B 0,C 180,E1 -24969.156,E2 -24969.156} C_VEL
LIN {X 0,Y 152.902,Z 651.414,A -85,B 0,C 180,E1 -24974.503,E2 -24974.503} C_VEL
LIN {X 0,Y 161.117,Z 642,A -85,B 0,C 180,E1 -24978.825,E2 -24978.825} C_VEL
LIN {X 0,Y 169.032,Z 632.384,A -85,B 0,C 180,E1 -24982.183,E2 -24982.183} C_VEL
LIN {X 0,Y 177.482,Z 621.151,A -85,B 0,C 180,E1 -24985.252,E2 -24985.252} C_VEL
LIN {X 0,Y 185.652,Z 609.195,A -85,B 0,C 180,E1 -24987.751,E2 -24987.751} C_VEL
LIN {X 0,Y 193.165,Z 596.747,A -85,B 0,C 180,E1 -24989.78,E2 -24989.78} C_VEL
LIN {X 0,Y 200.692,Z 582.458,A -85,B 0,C 180,E1 -24991.623,E2 -24991.623} C_VEL
LIN {X 0,Y 207.059,Z 568.563,A -85,B 0,C 180,E1 -24992.996,E2 -24992.996} C_VEL
LIN {X 0,Y 213.126,Z 552.546,A -85,B 0,C 180,E1 -24994.243,E2 -24994.243} C_VEL
LIN {X 0,Y 217.646,Z 537.622,A -85,B 0,C 180,E1 -24995.117,E2 -24995.117} C_VEL
LIN {X 0,Y 221.599,Z 521.191,A -85,B 0,C 180,E1 -24995.778,E2 -24995.778} C_VEL
LIN {X 0,Y 224.281,Z 504.501,A -85,B 0,C 180,E1 -24996.31,E2 -24996.31} C_VEL
LIN {X 0,Y 230.904,Z 435.757,A -85,B 0,C 180,E1 -24997.908,E2 -24997.908} C_VEL
LIN {X 0,Y 228.609,Z 429.699,A -85,B 0,C 180,E1 -24999.884,E2 -24999.884} C_VEL
LIN {X 0,Y 225.173,Z 422.776,A -85,B 0,C 180,E1 -25003.111,E2 -25003.111} C_VEL
LIN {X 0,Y 222.12,Z 416.956,A -85,B 0,C 180,E1 -25006.652,E2 -25006.652} C_VEL
LIN {X 0,Y 220.108,Z 413.241,A -85,B 0,C 180,E1 -25009.654,E2 -25009.654} C_VEL
LIN {X 0,Y 218.311,Z 409.566,A -85,B 0,C 180,E1 -25013.531,E2 -25013.531} C_VEL
LIN {X 0,Y 217.101,Z 407.304,A -85,B 0,C 180,E1 -25020,E2 -25020} C_VEL
LIN {X 0,Y 218.441,Z 409.829,A -85,B 0,C 180,E1 -25027.278,E2 -25027.278} C_VEL
LIN {X 0,Y 220.598,Z 414.169,A -85,B 0,C 180,E1 -25031.614,E2 -25031.614} C_VEL
LIN {X 0,Y 222.747,Z 418.241,A -85,B 0,C 180,E1 -25034.621,E2 -25034.621} C_VEL
LIN {X 0,Y 224.877,Z 422.216,A -85,B 0,C 180,E1 -25037.038,E2 -25037.038} C_VEL
LIN {X 0,Y 228.629,Z 429.69,A -85,B 0,C 180,E1 -25040.585,E2 -25040.585} C_VEL
LIN {X 0,Y 230.894,Z 434.563,A -85,B 0,C 180,E1 -25042.445,E2 -25042.445} C_VEL
LIN {X 0,Y 224.681,Z 499.87,A -85,B 0,C 180,E1 -25044.028,E2 -25044.028} C_VEL
LIN {X 0,Y 221.954,Z 516.606,A -85,B 0,C 180,E1 -25044.584,E2 -25044.584} C_VEL
LIN {X 0,Y 218.205,Z 532.66,A -85,B 0,C 180,E1 -25045.333,E2 -25045.333} C_VEL
LIN {X 0,Y 213.617,Z 547.922,A -85,B 0,C 180,E1 -25046.296,E2 -25046.296} C_VEL
LIN {X 0,Y 208.006,Z 562.863,A -85,B 0,C 180,E1 -25047.512,E2 -25047.512} C_VEL
LIN {X 0,Y 201.83,Z 576.696,A -85,B 0,C 180,E1 -25048.969,E2 -25048.969} C_VEL
LIN {X 0,Y 194.474,Z 590.891,A -85,B 0,C 180,E1 -25050.876,E2 -25050.876} C_VEL
LIN {X 0,Y 186.611,Z 603.953,A -85,B 0,C 180,E1 -25053.075,E2 -25053.075} C_VEL
LIN {X 0,Y 179.15,Z 615.078,A -85,B 0,C 180,E1 -25055.51,E2 -25055.51} C_VEL
LIN {X 0,Y 172.022,Z 624.666,A -85,B 0,C 180,E1 -25058.121,E2 -25058.121} C_VEL
LIN {X 0,Y 164.096,Z 634.461,A -85,B 0,C 180,E1 -25061.453,E2 -25061.453} C_VEL
LIN {X 0,Y 155.707,Z 643.827,A -85,B 0,C 180,E1 -25065.605,E2 -25065.605} C_VEL
LIN {X 0,Y 148.305,Z 651.655,A -85,B 0,C 180,E1 -25070.227,E2 -25070.227} C_VEL
LIN {X 0,Y 141.796,Z 658.182,A -85,B 0,C 180,E1 -25075.251,E2 -25075.251} C_VEL
LIN {X 0,Y 136.3,Z 663.578,A -85,B 0,C 180,E1 -25080.839,E2 -25080.839} C_VEL
LIN {X 0,Y 133.117,Z 666.71,A -85,B 0,C 180,E1 -25085.016,E2 -25085.016} C_VEL
LIN {X 0,Y 129.728,Z 670.05,A -85,B 0,C 180,E1 -25091.031,E2 -25091.031} C_VEL
LIN {X 0,Y 127.682,Z 672.467,A -85,B 0,C 180,E1 -25097.281,E2 -25097.281} C_VEL
LIN {X 0,Y 126.657,Z 673.83,A -85,B 0,C 180,E1 -25103.628,E2 -25103.628} C_VEL
LIN {X 0,Y 126.505,Z 674.349,A -85,B 0,C 180,E1 -25110,E2 -25110} C_VEL
LIN {X 0,Y 126.657,Z 673.86,A -85,B 0,C 180,E1 -25116.371,E2 -25116.371} C_VEL
LIN {X 0,Y 127.674,Z 672.526,A -85,B 0,C 180,E1 -25122.72,E2 -25122.72} C_VEL
LIN {X 0,Y 129.696,Z 670.138,A -85,B 0,C 180,E1 -25128.973,E2 -25128.973} C_VEL
LIN {X 0,Y 133.061,Z 666.834,A -85,B 0,C 180,E1 -25134.995,E2 -25134.995} C_VEL
LIN {X 0,Y 138.933,Z 661.149,A -85,B 0,C 180,E1 -25142.083,E2 -25142.083} C_VEL
LIN {X 0,Y 146.533,Z 653.656,A -85,B 0,C 180,E1 -25148.572,E2 -25148.572} C_VEL
LIN {X 0,Y 154.671,Z 645.163,A -85,B 0,C 180,E1 -25153.862,E2 -25153.862} C_VEL
LIN {X 0,Y 162.909,Z 635.982,A -85,B 0,C 180,E1 -25158.088,E2 -25158.088} C_VEL
LIN {X 0,Y 170.763,Z 626.525,A -85,B 0,C 180,E1 -25161.441,E2 -25161.441} C_VEL
LIN {X 0,Y 177.826,Z 617.192,A -85,B 0,C 180,E1 -25164.114,E2 -25164.114} C_VEL
LIN {X 0,Y 185.267,Z 606.349,A -85,B 0,C 180,E1 -25166.569,E2 -25166.569} C_VEL
LIN {X 0,Y 193.105,Z 593.77,A -85,B 0,C 180,E1 -25168.789,E2 -25168.789} C_VEL
LIN {X 0,Y 199.919,Z 581.033,A -85,B 0,C 180,E1 -25170.65,E2 -25170.65} C_VEL
LIN {X 0,Y 206.535,Z 566.879,A -85,B 0,C 180,E1 -25172.218,E2 -25172.218} C_VEL
LIN {X 0,Y 212.142,Z 552.801,A -85,B 0,C 180,E1 -25173.44,E2 -25173.44} C_VEL
LIN {X 0,Y 217.025,Z 537.745,A -85,B 0,C 180,E1 -25174.512,E2 -25174.512} C_VEL
LIN {X 0,Y 221.115,Z 521.67,A -85,B 0,C 180,E1 -25175.345,E2 -25175.345} C_VEL
LIN {X 0,Y 224.035,Z 505.782,A -85,B 0,C 180,E1 -25175.943,E2 -25175.943} C_VEL
LIN {X 0,Y 226.478,Z 484.566,A -85,B 0,C 180,E1 -25176.474,E2 -25176.474} C_VEL
LIN {X 0,Y 231.132,Z 434.793,A -85,B 0,C 180,E1 -25177.652,E2 -25177.652} C_VEL
LIN {X 0,Y 227.454,Z 427.001,A -85,B 0,C 180,E1 -25180.776,E2 -25180.776} C_VEL
LIN {X 0,Y 224.125,Z 420.463,A -85,B 0,C 180,E1 -25184.162,E2 -25184.162} C_VEL
LIN {X 0,Y 221.874,Z 416.416,A -85,B 0,C 180,E1 -25186.956,E2 -25186.956} C_VEL
LIN {X 0,Y 220.295,Z 413.354,A -85,B 0,C 180,E1 -25189.43,E2 -25189.43} C_VEL
LIN {X 0,Y 218.455,Z 409.612,A -85,B 0,C 180,E1 -25193.535,E2 -25193.535} C_VEL
LIN {X 0,Y 217.378,Z 407.708,A -85,B 0,C 180,E1 -25200,E2 -25200} C_VEL
LIN {X 0,Y 218.664,Z 410.03,A -85,B 0,C 180,E1 -25206.69,E2 -25206.69} C_VEL
LIN {X 0,Y 220.372,Z 413.466,A -85,B 0,C 180,E1 -25210.334,E2 -25210.334} C_VEL
LIN {X 0,Y 222.895,Z 418.316,A -85,B 0,C 180,E1 -25214.027,E2 -25214.027} C_VEL
LIN {X 0,Y 225.633,Z 423.395,A -85,B 0,C 180,E1 -25217.095,E2 -25217.095} C_VEL
LIN {X 0,Y 229.141,Z 430.572,A -85,B 0,C 180,E1 -25220.36,E2 -25220.36} C_VEL
LIN {X 0,Y 231.143,Z 435.932,A -85,B 0,C 180,E1 -25222.081,E2 -25222.081} C_VEL
LIN {X 0,Y 224.135,Z 507.665,A -85,B 0,C 180,E1 -25223.746,E2 -25223.746} C_VEL
LIN {X 0,Y 221.311,Z 523.659,A -85,B 0,C 180,E1 -25224.269,E2 -25224.269} C_VEL
LIN {X 0,Y 217.527,Z 539,A -85,B 0,C 180,E1 -25224.946,E2 -25224.946} C_VEL
LIN {X 0,Y 212.75,Z 554.139,A -85,B 0,C 180,E1 -25225.82,E2 -25225.82} C_VEL
LIN {X 0,Y 207.025,Z 569.077,A -85,B 0,C 180,E1 -25226.986,E2 -25226.986} C_VEL
LIN {X 0,Y 200.013,Z 584.301,A -85,B 0,C 180,E1 -25228.546,E2 -25228.546} C_VEL
LIN {X 0,Y 193.163,Z 597.081,A -85,B 0,C 180,E1 -25230.219,E2 -25230.219} C_VEL
LIN {X 0,Y 190.621,Z 601.516,A -85,B 0,C 180,E1 -25230.891,E2 -25230.891} C_VEL
LIN {X 0,Y 187.435,Z 606.132,A -85,B 0,C 180,E1 -25231.467,E2 -25231.467} C_VEL
LIN {X 0,Y 181.039,Z 613.478,A -85,B 0,C 180,E1 -25232.076,E2 -25232.076} C_VEL
LIN {X 0,Y 174.433,Z 620.496,A -85,B 0,C 180,E1 -25232.827,E2 -25232.827} C_VEL
LIN {X 0,Y 170.959,Z 624.557,A -85,B 0,C 180,E1 -25233.648,E2 -25233.648} C_VEL
LIN {X 0,Y 162.33,Z 635.317,A -85,B 0,C 180,E1 -25236.78,E2 -25236.78} C_VEL
LIN {X 0,Y 154.34,Z 644.478,A -85,B 0,C 180,E1 -25240.296,E2 -25240.296} C_VEL
LIN {X 0,Y 145.79,Z 653.379,A -85,B 0,C 180,E1 -25244.681,E2 -25244.681} C_VEL
LIN {X 0,Y 138.137,Z 661.013,A -85,B 0,C 180,E1 -25249.742,E2 -25249.742} C_VEL
LIN {X 0,Y 131.2,Z 667.72,A -85,B 0,C 180,E1 -25255.775,E2 -25255.775} C_VEL
LIN {X 0,Y 125.196,Z 673.594,A -85,B 0,C 180,E1 -25263.315,E2 -25263.315} C_VEL
LIN {X 0,Y 121.858,Z 677.038,A -85,B 0,C 180,E1 -25269.755,E2 -25269.755} C_VEL
LIN {X 0,Y 119.851,Z 679.552,A -85,B 0,C 180,E1 -25276.435,E2 -25276.435} C_VEL
LIN {X 0,Y 119.168,Z 680.983,A -85,B 0,C 180,E1 -25283.226,E2 -25283.226} C_VEL
LIN {X 0,Y 119.332,Z 681.527,A -85,B 0,C 180,E1 -25290,E2 -25290} C_VEL
LIN {X 0,Y 119.168,Z 680.967,A -85,B 0,C 180,E1 -25296.774,E2 -25296.774} C_VEL
LIN {X 0,Y 119.851,Z 679.518,A -85,B 0,C 180,E1 -25303.566,E2 -25303.566} C_VEL
LIN {X 0,Y 121.853,Z 676.989,A -85,B 0,C 180,E1 -25310.246,E2 -25310.246} C_VEL
LIN {X 0,Y 125.196,Z 673.527,A -85,B 0,C 180,E1 -25316.685,E2 -25316.685} C_VEL
LIN {X 0,Y 131.216,Z 667.631,A -85,B 0,C 180,E1 -25324.221,E2 -25324.221} C_VEL
LIN {X 0,Y 139.175,Z 659.901,A -85,B 0,C 180,E1 -25331.031,E2 -25331.031} C_VEL
LIN {X 0,Y 147.839,Z 651.202,A -85,B 0,C 180,E1 -25336.465,E2 -25336.465} C_VEL
LIN {X 0,Y 155.32,Z 643.058,A -85,B 0,C 180,E1 -25340.284,E2 -25340.284} C_VEL
LIN {X 0,Y 164.719,Z 632.171,A -85,B 0,C 180,E1 -25344.161,E2 -25344.161} C_VEL
LIN {X 0,Y 173.491,Z 620.939,A -85,B 0,C 180,E1 -25347.2,E2 -25347.2} C_VEL
LIN {X 0,Y 181.678,Z 609.347,A -85,B 0,C 180,E1 -25349.591,E2 -25349.591} C_VEL
LIN {X 0,Y 189.664,Z 596.534,A -85,B 0,C 180,E1 -25351.648,E2 -25351.648} C_VEL
LIN {X 0,Y 197.409,Z 582.246,A -85,B 0,C 180,E1 -25353.441,E2 -25353.441} C_VEL
LIN {X 0,Y 203.928,Z 568.35,A -85,B 0,C 180,E1 -25354.776,E2 -25354.776} C_VEL
LIN {X 0,Y 209.76,Z 553.343,A -85,B 0,C 180,E1 -25355.924,E2 -25355.924} C_VEL
LIN {X 0,Y 214.551,Z 538.09,A -85,B 0,C 180,E1 -25356.807,E2 -25356.807} C_VEL
LIN {X 0,Y 218.749,Z 521.13,A -85,B 0,C 180,E1 -25357.469,E2 -25357.469} C_VEL
